;FOLD LIN P827 Vel=2 m/s CPDAT827 Tool[1]:marker Base[0] ;%{PE}
;FOLD Parameters ;%{h}
;Params IlfProvider=kukaroboter.basistech.inlineforms.movement.old; Kuka.IsGlobalPoint=False; Kuka.PointName=P827; Kuka.BlendingEnabled=False; Kuka.MoveDataName=CPDAT1; Kuka.VelocityPath=2; Kuka.CurrentCDSetIndex=0; Kuka.MovementParameterFieldEnabled=True; IlfCommand=LIN
;ENDFOLD
$BWDSTART = FALSE
LDAT_ACT = LCPDAT827
FDAT_ACT = FP827
BAS(#CP_PARAMS, 2.0)
SET_CD_PARAMS (0)
LIN XP827
;ENDFOLD

;FOLD LIN P828 Vel=2 m/s CPDAT828 Tool[1]:marker Base[0] ;%{PE}
;FOLD Parameters ;%{h}
;Params IlfProvider=kukaroboter.basistech.inlineforms.movement.old; Kuka.IsGlobalPoint=False; Kuka.PointName=P828; Kuka.BlendingEnabled=False; Kuka.MoveDataName=CPDAT1; Kuka.VelocityPath=2; Kuka.CurrentCDSetIndex=0; Kuka.MovementParameterFieldEnabled=True; IlfCommand=LIN
;ENDFOLD
$BWDSTART = FALSE
LDAT_ACT = LCPDAT828
FDAT_ACT = FP828
BAS(#CP_PARAMS, 2.0)
SET_CD_PARAMS (0)
LIN XP828
;ENDFOLD

;FOLD LIN P829 Vel=2 m/s CPDAT829 Tool[1]:marker Base[0] ;%{PE}
;FOLD Parameters ;%{h}
;Params IlfProvider=kukaroboter.basistech.inlineforms.movement.old; Kuka.IsGlobalPoint=False; Kuka.PointName=P829; Kuka.BlendingEnabled=False; Kuka.MoveDataName=CPDAT1; Kuka.VelocityPath=2; Kuka.CurrentCDSetIndex=0; Kuka.MovementParameterFieldEnabled=True; IlfCommand=LIN
;ENDFOLD
$BWDSTART = FALSE
LDAT_ACT = LCPDAT829
FDAT_ACT = FP829
BAS(#CP_PARAMS, 2.0)
SET_CD_PARAMS (0)
LIN XP829
;ENDFOLD

;FOLD LIN P830 Vel=2 m/s CPDAT830 Tool[1]:marker Base[0] ;%{PE}
;FOLD Parameters ;%{h}
;Params IlfProvider=kukaroboter.basistech.inlineforms.movement.old; Kuka.IsGlobalPoint=False; Kuka.PointName=P830; Kuka.BlendingEnabled=False; Kuka.MoveDataName=CPDAT1; Kuka.VelocityPath=2; Kuka.CurrentCDSetIndex=0; Kuka.MovementParameterFieldEnabled=True; IlfCommand=LIN
;ENDFOLD
$BWDSTART = FALSE
LDAT_ACT = LCPDAT830
FDAT_ACT = FP830
BAS(#CP_PARAMS, 2.0)
SET_CD_PARAMS (0)
LIN XP830
;ENDFOLD

;FOLD LIN P831 Vel=2 m/s CPDAT831 Tool[1]:marker Base[0] ;%{PE}
;FOLD Parameters ;%{h}
;Params IlfProvider=kukaroboter.basistech.inlineforms.movement.old; Kuka.IsGlobalPoint=False; Kuka.PointName=P831; Kuka.BlendingEnabled=False; Kuka.MoveDataName=CPDAT1; Kuka.VelocityPath=2; Kuka.CurrentCDSetIndex=0; Kuka.MovementParameterFieldEnabled=True; IlfCommand=LIN
;ENDFOLD
$BWDSTART = FALSE
LDAT_ACT = LCPDAT831
FDAT_ACT = FP831
BAS(#CP_PARAMS, 2.0)
SET_CD_PARAMS (0)
LIN XP831
;ENDFOLD

;FOLD LIN P832 Vel=2 m/s CPDAT832 Tool[1]:marker Base[0] ;%{PE}
;FOLD Parameters ;%{h}
;Params IlfProvider=kukaroboter.basistech.inlineforms.movement.old; Kuka.IsGlobalPoint=False; Kuka.PointName=P832; Kuka.BlendingEnabled=False; Kuka.MoveDataName=CPDAT1; Kuka.VelocityPath=2; Kuka.CurrentCDSetIndex=0; Kuka.MovementParameterFieldEnabled=True; IlfCommand=LIN
;ENDFOLD
$BWDSTART = FALSE
LDAT_ACT = LCPDAT832
FDAT_ACT = FP832
BAS(#CP_PARAMS, 2.0)
SET_CD_PARAMS (0)
LIN XP832
;ENDFOLD

;FOLD LIN P833 Vel=2 m/s CPDAT833 Tool[1]:marker Base[0] ;%{PE}
;FOLD Parameters ;%{h}
;Params IlfProvider=kukaroboter.basistech.inlineforms.movement.old; Kuka.IsGlobalPoint=False; Kuka.PointName=P833; Kuka.BlendingEnabled=False; Kuka.MoveDataName=CPDAT1; Kuka.VelocityPath=2; Kuka.CurrentCDSetIndex=0; Kuka.MovementParameterFieldEnabled=True; IlfCommand=LIN
;ENDFOLD
$BWDSTART = FALSE
LDAT_ACT = LCPDAT833
FDAT_ACT = FP833
BAS(#CP_PARAMS, 2.0)
SET_CD_PARAMS (0)
LIN XP833
;ENDFOLD

;FOLD LIN P834 Vel=2 m/s CPDAT834 Tool[1]:marker Base[0] ;%{PE}
;FOLD Parameters ;%{h}
;Params IlfProvider=kukaroboter.basistech.inlineforms.movement.old; Kuka.IsGlobalPoint=False; Kuka.PointName=P834; Kuka.BlendingEnabled=False; Kuka.MoveDataName=CPDAT1; Kuka.VelocityPath=2; Kuka.CurrentCDSetIndex=0; Kuka.MovementParameterFieldEnabled=True; IlfCommand=LIN
;ENDFOLD
$BWDSTART = FALSE
LDAT_ACT = LCPDAT834
FDAT_ACT = FP834
BAS(#CP_PARAMS, 2.0)
SET_CD_PARAMS (0)
LIN XP834
;ENDFOLD

;FOLD LIN P835 Vel=2 m/s CPDAT835 Tool[1]:marker Base[0] ;%{PE}
;FOLD Parameters ;%{h}
;Params IlfProvider=kukaroboter.basistech.inlineforms.movement.old; Kuka.IsGlobalPoint=False; Kuka.PointName=P835; Kuka.BlendingEnabled=False; Kuka.MoveDataName=CPDAT1; Kuka.VelocityPath=2; Kuka.CurrentCDSetIndex=0; Kuka.MovementParameterFieldEnabled=True; IlfCommand=LIN
;ENDFOLD
$BWDSTART = FALSE
LDAT_ACT = LCPDAT835
FDAT_ACT = FP835
BAS(#CP_PARAMS, 2.0)
SET_CD_PARAMS (0)
LIN XP835
;ENDFOLD

;FOLD LIN P836 Vel=2 m/s CPDAT836 Tool[1]:marker Base[0] ;%{PE}
;FOLD Parameters ;%{h}
;Params IlfProvider=kukaroboter.basistech.inlineforms.movement.old; Kuka.IsGlobalPoint=False; Kuka.PointName=P836; Kuka.BlendingEnabled=False; Kuka.MoveDataName=CPDAT1; Kuka.VelocityPath=2; Kuka.CurrentCDSetIndex=0; Kuka.MovementParameterFieldEnabled=True; IlfCommand=LIN
;ENDFOLD
$BWDSTART = FALSE
LDAT_ACT = LCPDAT836
FDAT_ACT = FP836
BAS(#CP_PARAMS, 2.0)
SET_CD_PARAMS (0)
LIN XP836
;ENDFOLD

;FOLD LIN P837 Vel=2 m/s CPDAT837 Tool[1]:marker Base[0] ;%{PE}
;FOLD Parameters ;%{h}
;Params IlfProvider=kukaroboter.basistech.inlineforms.movement.old; Kuka.IsGlobalPoint=False; Kuka.PointName=P837; Kuka.BlendingEnabled=False; Kuka.MoveDataName=CPDAT1; Kuka.VelocityPath=2; Kuka.CurrentCDSetIndex=0; Kuka.MovementParameterFieldEnabled=True; IlfCommand=LIN
;ENDFOLD
$BWDSTART = FALSE
LDAT_ACT = LCPDAT837
FDAT_ACT = FP837
BAS(#CP_PARAMS, 2.0)
SET_CD_PARAMS (0)
LIN XP837
;ENDFOLD

;FOLD LIN P838 Vel=2 m/s CPDAT838 Tool[1]:marker Base[0] ;%{PE}
;FOLD Parameters ;%{h}
;Params IlfProvider=kukaroboter.basistech.inlineforms.movement.old; Kuka.IsGlobalPoint=False; Kuka.PointName=P838; Kuka.BlendingEnabled=False; Kuka.MoveDataName=CPDAT1; Kuka.VelocityPath=2; Kuka.CurrentCDSetIndex=0; Kuka.MovementParameterFieldEnabled=True; IlfCommand=LIN
;ENDFOLD
$BWDSTART = FALSE
LDAT_ACT = LCPDAT838
FDAT_ACT = FP838
BAS(#CP_PARAMS, 2.0)
SET_CD_PARAMS (0)
LIN XP838
;ENDFOLD

;FOLD LIN P839 Vel=2 m/s CPDAT839 Tool[1]:marker Base[0] ;%{PE}
;FOLD Parameters ;%{h}
;Params IlfProvider=kukaroboter.basistech.inlineforms.movement.old; Kuka.IsGlobalPoint=False; Kuka.PointName=P839; Kuka.BlendingEnabled=False; Kuka.MoveDataName=CPDAT1; Kuka.VelocityPath=2; Kuka.CurrentCDSetIndex=0; Kuka.MovementParameterFieldEnabled=True; IlfCommand=LIN
;ENDFOLD
$BWDSTART = FALSE
LDAT_ACT = LCPDAT839
FDAT_ACT = FP839
BAS(#CP_PARAMS, 2.0)
SET_CD_PARAMS (0)
LIN XP839
;ENDFOLD

;FOLD LIN P840 Vel=2 m/s CPDAT840 Tool[1]:marker Base[0] ;%{PE}
;FOLD Parameters ;%{h}
;Params IlfProvider=kukaroboter.basistech.inlineforms.movement.old; Kuka.IsGlobalPoint=False; Kuka.PointName=P840; Kuka.BlendingEnabled=False; Kuka.MoveDataName=CPDAT1; Kuka.VelocityPath=2; Kuka.CurrentCDSetIndex=0; Kuka.MovementParameterFieldEnabled=True; IlfCommand=LIN
;ENDFOLD
$BWDSTART = FALSE
LDAT_ACT = LCPDAT840
FDAT_ACT = FP840
BAS(#CP_PARAMS, 2.0)
SET_CD_PARAMS (0)
LIN XP840
;ENDFOLD

;FOLD LIN P841 Vel=2 m/s CPDAT841 Tool[1]:marker Base[0] ;%{PE}
;FOLD Parameters ;%{h}
;Params IlfProvider=kukaroboter.basistech.inlineforms.movement.old; Kuka.IsGlobalPoint=False; Kuka.PointName=P841; Kuka.BlendingEnabled=False; Kuka.MoveDataName=CPDAT1; Kuka.VelocityPath=2; Kuka.CurrentCDSetIndex=0; Kuka.MovementParameterFieldEnabled=True; IlfCommand=LIN
;ENDFOLD
$BWDSTART = FALSE
LDAT_ACT = LCPDAT841
FDAT_ACT = FP841
BAS(#CP_PARAMS, 2.0)
SET_CD_PARAMS (0)
LIN XP841
;ENDFOLD

;FOLD LIN P842 Vel=2 m/s CPDAT842 Tool[1]:marker Base[0] ;%{PE}
;FOLD Parameters ;%{h}
;Params IlfProvider=kukaroboter.basistech.inlineforms.movement.old; Kuka.IsGlobalPoint=False; Kuka.PointName=P842; Kuka.BlendingEnabled=False; Kuka.MoveDataName=CPDAT1; Kuka.VelocityPath=2; Kuka.CurrentCDSetIndex=0; Kuka.MovementParameterFieldEnabled=True; IlfCommand=LIN
;ENDFOLD
$BWDSTART = FALSE
LDAT_ACT = LCPDAT842
FDAT_ACT = FP842
BAS(#CP_PARAMS, 2.0)
SET_CD_PARAMS (0)
LIN XP842
;ENDFOLD

;FOLD LIN P843 Vel=2 m/s CPDAT843 Tool[1]:marker Base[0] ;%{PE}
;FOLD Parameters ;%{h}
;Params IlfProvider=kukaroboter.basistech.inlineforms.movement.old; Kuka.IsGlobalPoint=False; Kuka.PointName=P843; Kuka.BlendingEnabled=False; Kuka.MoveDataName=CPDAT1; Kuka.VelocityPath=2; Kuka.CurrentCDSetIndex=0; Kuka.MovementParameterFieldEnabled=True; IlfCommand=LIN
;ENDFOLD
$BWDSTART = FALSE
LDAT_ACT = LCPDAT843
FDAT_ACT = FP843
BAS(#CP_PARAMS, 2.0)
SET_CD_PARAMS (0)
LIN XP843
;ENDFOLD

;FOLD LIN P844 Vel=2 m/s CPDAT844 Tool[1]:marker Base[0] ;%{PE}
;FOLD Parameters ;%{h}
;Params IlfProvider=kukaroboter.basistech.inlineforms.movement.old; Kuka.IsGlobalPoint=False; Kuka.PointName=P844; Kuka.BlendingEnabled=False; Kuka.MoveDataName=CPDAT1; Kuka.VelocityPath=2; Kuka.CurrentCDSetIndex=0; Kuka.MovementParameterFieldEnabled=True; IlfCommand=LIN
;ENDFOLD
$BWDSTART = FALSE
LDAT_ACT = LCPDAT844
FDAT_ACT = FP844
BAS(#CP_PARAMS, 2.0)
SET_CD_PARAMS (0)
LIN XP844
;ENDFOLD

;FOLD LIN P845 Vel=2 m/s CPDAT845 Tool[1]:marker Base[0] ;%{PE}
;FOLD Parameters ;%{h}
;Params IlfProvider=kukaroboter.basistech.inlineforms.movement.old; Kuka.IsGlobalPoint=False; Kuka.PointName=P845; Kuka.BlendingEnabled=False; Kuka.MoveDataName=CPDAT1; Kuka.VelocityPath=2; Kuka.CurrentCDSetIndex=0; Kuka.MovementParameterFieldEnabled=True; IlfCommand=LIN
;ENDFOLD
$BWDSTART = FALSE
LDAT_ACT = LCPDAT845
FDAT_ACT = FP845
BAS(#CP_PARAMS, 2.0)
SET_CD_PARAMS (0)
LIN XP845
;ENDFOLD

;FOLD LIN P846 Vel=2 m/s CPDAT846 Tool[1]:marker Base[0] ;%{PE}
;FOLD Parameters ;%{h}
;Params IlfProvider=kukaroboter.basistech.inlineforms.movement.old; Kuka.IsGlobalPoint=False; Kuka.PointName=P846; Kuka.BlendingEnabled=False; Kuka.MoveDataName=CPDAT1; Kuka.VelocityPath=2; Kuka.CurrentCDSetIndex=0; Kuka.MovementParameterFieldEnabled=True; IlfCommand=LIN
;ENDFOLD
$BWDSTART = FALSE
LDAT_ACT = LCPDAT846
FDAT_ACT = FP846
BAS(#CP_PARAMS, 2.0)
SET_CD_PARAMS (0)
LIN XP846
;ENDFOLD

;FOLD LIN P847 Vel=2 m/s CPDAT847 Tool[1]:marker Base[0] ;%{PE}
;FOLD Parameters ;%{h}
;Params IlfProvider=kukaroboter.basistech.inlineforms.movement.old; Kuka.IsGlobalPoint=False; Kuka.PointName=P847; Kuka.BlendingEnabled=False; Kuka.MoveDataName=CPDAT1; Kuka.VelocityPath=2; Kuka.CurrentCDSetIndex=0; Kuka.MovementParameterFieldEnabled=True; IlfCommand=LIN
;ENDFOLD
$BWDSTART = FALSE
LDAT_ACT = LCPDAT847
FDAT_ACT = FP847
BAS(#CP_PARAMS, 2.0)
SET_CD_PARAMS (0)
LIN XP847
;ENDFOLD

;FOLD LIN P848 Vel=2 m/s CPDAT848 Tool[1]:marker Base[0] ;%{PE}
;FOLD Parameters ;%{h}
;Params IlfProvider=kukaroboter.basistech.inlineforms.movement.old; Kuka.IsGlobalPoint=False; Kuka.PointName=P848; Kuka.BlendingEnabled=False; Kuka.MoveDataName=CPDAT1; Kuka.VelocityPath=2; Kuka.CurrentCDSetIndex=0; Kuka.MovementParameterFieldEnabled=True; IlfCommand=LIN
;ENDFOLD
$BWDSTART = FALSE
LDAT_ACT = LCPDAT848
FDAT_ACT = FP848
BAS(#CP_PARAMS, 2.0)
SET_CD_PARAMS (0)
LIN XP848
;ENDFOLD

;FOLD LIN P849 Vel=2 m/s CPDAT849 Tool[1]:marker Base[0] ;%{PE}
;FOLD Parameters ;%{h}
;Params IlfProvider=kukaroboter.basistech.inlineforms.movement.old; Kuka.IsGlobalPoint=False; Kuka.PointName=P849; Kuka.BlendingEnabled=False; Kuka.MoveDataName=CPDAT1; Kuka.VelocityPath=2; Kuka.CurrentCDSetIndex=0; Kuka.MovementParameterFieldEnabled=True; IlfCommand=LIN
;ENDFOLD
$BWDSTART = FALSE
LDAT_ACT = LCPDAT849
FDAT_ACT = FP849
BAS(#CP_PARAMS, 2.0)
SET_CD_PARAMS (0)
LIN XP849
;ENDFOLD

;FOLD LIN P850 Vel=2 m/s CPDAT850 Tool[1]:marker Base[0] ;%{PE}
;FOLD Parameters ;%{h}
;Params IlfProvider=kukaroboter.basistech.inlineforms.movement.old; Kuka.IsGlobalPoint=False; Kuka.PointName=P850; Kuka.BlendingEnabled=False; Kuka.MoveDataName=CPDAT1; Kuka.VelocityPath=2; Kuka.CurrentCDSetIndex=0; Kuka.MovementParameterFieldEnabled=True; IlfCommand=LIN
;ENDFOLD
$BWDSTART = FALSE
LDAT_ACT = LCPDAT850
FDAT_ACT = FP850
BAS(#CP_PARAMS, 2.0)
SET_CD_PARAMS (0)
LIN XP850
;ENDFOLD

;FOLD LIN P851 Vel=2 m/s CPDAT851 Tool[1]:marker Base[0] ;%{PE}
;FOLD Parameters ;%{h}
;Params IlfProvider=kukaroboter.basistech.inlineforms.movement.old; Kuka.IsGlobalPoint=False; Kuka.PointName=P851; Kuka.BlendingEnabled=False; Kuka.MoveDataName=CPDAT1; Kuka.VelocityPath=2; Kuka.CurrentCDSetIndex=0; Kuka.MovementParameterFieldEnabled=True; IlfCommand=LIN
;ENDFOLD
$BWDSTART = FALSE
LDAT_ACT = LCPDAT851
FDAT_ACT = FP851
BAS(#CP_PARAMS, 2.0)
SET_CD_PARAMS (0)
LIN XP851
;ENDFOLD

;FOLD LIN P852 Vel=2 m/s CPDAT852 Tool[1]:marker Base[0] ;%{PE}
;FOLD Parameters ;%{h}
;Params IlfProvider=kukaroboter.basistech.inlineforms.movement.old; Kuka.IsGlobalPoint=False; Kuka.PointName=P852; Kuka.BlendingEnabled=False; Kuka.MoveDataName=CPDAT1; Kuka.VelocityPath=2; Kuka.CurrentCDSetIndex=0; Kuka.MovementParameterFieldEnabled=True; IlfCommand=LIN
;ENDFOLD
$BWDSTART = FALSE
LDAT_ACT = LCPDAT852
FDAT_ACT = FP852
BAS(#CP_PARAMS, 2.0)
SET_CD_PARAMS (0)
LIN XP852
;ENDFOLD

;FOLD LIN P853 Vel=2 m/s CPDAT853 Tool[1]:marker Base[0] ;%{PE}
;FOLD Parameters ;%{h}
;Params IlfProvider=kukaroboter.basistech.inlineforms.movement.old; Kuka.IsGlobalPoint=False; Kuka.PointName=P853; Kuka.BlendingEnabled=False; Kuka.MoveDataName=CPDAT1; Kuka.VelocityPath=2; Kuka.CurrentCDSetIndex=0; Kuka.MovementParameterFieldEnabled=True; IlfCommand=LIN
;ENDFOLD
$BWDSTART = FALSE
LDAT_ACT = LCPDAT853
FDAT_ACT = FP853
BAS(#CP_PARAMS, 2.0)
SET_CD_PARAMS (0)
LIN XP853
;ENDFOLD

;FOLD LIN P854 Vel=2 m/s CPDAT854 Tool[1]:marker Base[0] ;%{PE}
;FOLD Parameters ;%{h}
;Params IlfProvider=kukaroboter.basistech.inlineforms.movement.old; Kuka.IsGlobalPoint=False; Kuka.PointName=P854; Kuka.BlendingEnabled=False; Kuka.MoveDataName=CPDAT1; Kuka.VelocityPath=2; Kuka.CurrentCDSetIndex=0; Kuka.MovementParameterFieldEnabled=True; IlfCommand=LIN
;ENDFOLD
$BWDSTART = FALSE
LDAT_ACT = LCPDAT854
FDAT_ACT = FP854
BAS(#CP_PARAMS, 2.0)
SET_CD_PARAMS (0)
LIN XP854
;ENDFOLD

;FOLD LIN P855 Vel=2 m/s CPDAT855 Tool[1]:marker Base[0] ;%{PE}
;FOLD Parameters ;%{h}
;Params IlfProvider=kukaroboter.basistech.inlineforms.movement.old; Kuka.IsGlobalPoint=False; Kuka.PointName=P855; Kuka.BlendingEnabled=False; Kuka.MoveDataName=CPDAT1; Kuka.VelocityPath=2; Kuka.CurrentCDSetIndex=0; Kuka.MovementParameterFieldEnabled=True; IlfCommand=LIN
;ENDFOLD
$BWDSTART = FALSE
LDAT_ACT = LCPDAT855
FDAT_ACT = FP855
BAS(#CP_PARAMS, 2.0)
SET_CD_PARAMS (0)
LIN XP855
;ENDFOLD

;FOLD LIN P856 Vel=2 m/s CPDAT856 Tool[1]:marker Base[0] ;%{PE}
;FOLD Parameters ;%{h}
;Params IlfProvider=kukaroboter.basistech.inlineforms.movement.old; Kuka.IsGlobalPoint=False; Kuka.PointName=P856; Kuka.BlendingEnabled=False; Kuka.MoveDataName=CPDAT1; Kuka.VelocityPath=2; Kuka.CurrentCDSetIndex=0; Kuka.MovementParameterFieldEnabled=True; IlfCommand=LIN
;ENDFOLD
$BWDSTART = FALSE
LDAT_ACT = LCPDAT856
FDAT_ACT = FP856
BAS(#CP_PARAMS, 2.0)
SET_CD_PARAMS (0)
LIN XP856
;ENDFOLD

;FOLD LIN P857 Vel=2 m/s CPDAT857 Tool[1]:marker Base[0] ;%{PE}
;FOLD Parameters ;%{h}
;Params IlfProvider=kukaroboter.basistech.inlineforms.movement.old; Kuka.IsGlobalPoint=False; Kuka.PointName=P857; Kuka.BlendingEnabled=False; Kuka.MoveDataName=CPDAT1; Kuka.VelocityPath=2; Kuka.CurrentCDSetIndex=0; Kuka.MovementParameterFieldEnabled=True; IlfCommand=LIN
;ENDFOLD
$BWDSTART = FALSE
LDAT_ACT = LCPDAT857
FDAT_ACT = FP857
BAS(#CP_PARAMS, 2.0)
SET_CD_PARAMS (0)
LIN XP857
;ENDFOLD

;FOLD LIN P858 Vel=2 m/s CPDAT858 Tool[1]:marker Base[0] ;%{PE}
;FOLD Parameters ;%{h}
;Params IlfProvider=kukaroboter.basistech.inlineforms.movement.old; Kuka.IsGlobalPoint=False; Kuka.PointName=P858; Kuka.BlendingEnabled=False; Kuka.MoveDataName=CPDAT1; Kuka.VelocityPath=2; Kuka.CurrentCDSetIndex=0; Kuka.MovementParameterFieldEnabled=True; IlfCommand=LIN
;ENDFOLD
$BWDSTART = FALSE
LDAT_ACT = LCPDAT858
FDAT_ACT = FP858
BAS(#CP_PARAMS, 2.0)
SET_CD_PARAMS (0)
LIN XP858
;ENDFOLD

;FOLD LIN P859 Vel=2 m/s CPDAT859 Tool[1]:marker Base[0] ;%{PE}
;FOLD Parameters ;%{h}
;Params IlfProvider=kukaroboter.basistech.inlineforms.movement.old; Kuka.IsGlobalPoint=False; Kuka.PointName=P859; Kuka.BlendingEnabled=False; Kuka.MoveDataName=CPDAT1; Kuka.VelocityPath=2; Kuka.CurrentCDSetIndex=0; Kuka.MovementParameterFieldEnabled=True; IlfCommand=LIN
;ENDFOLD
$BWDSTART = FALSE
LDAT_ACT = LCPDAT859
FDAT_ACT = FP859
BAS(#CP_PARAMS, 2.0)
SET_CD_PARAMS (0)
LIN XP859
;ENDFOLD

;FOLD LIN P860 Vel=2 m/s CPDAT860 Tool[1]:marker Base[0] ;%{PE}
;FOLD Parameters ;%{h}
;Params IlfProvider=kukaroboter.basistech.inlineforms.movement.old; Kuka.IsGlobalPoint=False; Kuka.PointName=P860; Kuka.BlendingEnabled=False; Kuka.MoveDataName=CPDAT1; Kuka.VelocityPath=2; Kuka.CurrentCDSetIndex=0; Kuka.MovementParameterFieldEnabled=True; IlfCommand=LIN
;ENDFOLD
$BWDSTART = FALSE
LDAT_ACT = LCPDAT860
FDAT_ACT = FP860
BAS(#CP_PARAMS, 2.0)
SET_CD_PARAMS (0)
LIN XP860
;ENDFOLD

;FOLD LIN P861 Vel=2 m/s CPDAT861 Tool[1]:marker Base[0] ;%{PE}
;FOLD Parameters ;%{h}
;Params IlfProvider=kukaroboter.basistech.inlineforms.movement.old; Kuka.IsGlobalPoint=False; Kuka.PointName=P861; Kuka.BlendingEnabled=False; Kuka.MoveDataName=CPDAT1; Kuka.VelocityPath=2; Kuka.CurrentCDSetIndex=0; Kuka.MovementParameterFieldEnabled=True; IlfCommand=LIN
;ENDFOLD
$BWDSTART = FALSE
LDAT_ACT = LCPDAT861
FDAT_ACT = FP861
BAS(#CP_PARAMS, 2.0)
SET_CD_PARAMS (0)
LIN XP861
;ENDFOLD

;FOLD LIN P862 Vel=2 m/s CPDAT862 Tool[1]:marker Base[0] ;%{PE}
;FOLD Parameters ;%{h}
;Params IlfProvider=kukaroboter.basistech.inlineforms.movement.old; Kuka.IsGlobalPoint=False; Kuka.PointName=P862; Kuka.BlendingEnabled=False; Kuka.MoveDataName=CPDAT1; Kuka.VelocityPath=2; Kuka.CurrentCDSetIndex=0; Kuka.MovementParameterFieldEnabled=True; IlfCommand=LIN
;ENDFOLD
$BWDSTART = FALSE
LDAT_ACT = LCPDAT862
FDAT_ACT = FP862
BAS(#CP_PARAMS, 2.0)
SET_CD_PARAMS (0)
LIN XP862
;ENDFOLD

;FOLD LIN P863 Vel=2 m/s CPDAT863 Tool[1]:marker Base[0] ;%{PE}
;FOLD Parameters ;%{h}
;Params IlfProvider=kukaroboter.basistech.inlineforms.movement.old; Kuka.IsGlobalPoint=False; Kuka.PointName=P863; Kuka.BlendingEnabled=False; Kuka.MoveDataName=CPDAT1; Kuka.VelocityPath=2; Kuka.CurrentCDSetIndex=0; Kuka.MovementParameterFieldEnabled=True; IlfCommand=LIN
;ENDFOLD
$BWDSTART = FALSE
LDAT_ACT = LCPDAT863
FDAT_ACT = FP863
BAS(#CP_PARAMS, 2.0)
SET_CD_PARAMS (0)
LIN XP863
;ENDFOLD

;FOLD LIN P864 Vel=2 m/s CPDAT864 Tool[1]:marker Base[0] ;%{PE}
;FOLD Parameters ;%{h}
;Params IlfProvider=kukaroboter.basistech.inlineforms.movement.old; Kuka.IsGlobalPoint=False; Kuka.PointName=P864; Kuka.BlendingEnabled=False; Kuka.MoveDataName=CPDAT1; Kuka.VelocityPath=2; Kuka.CurrentCDSetIndex=0; Kuka.MovementParameterFieldEnabled=True; IlfCommand=LIN
;ENDFOLD
$BWDSTART = FALSE
LDAT_ACT = LCPDAT864
FDAT_ACT = FP864
BAS(#CP_PARAMS, 2.0)
SET_CD_PARAMS (0)
LIN XP864
;ENDFOLD

;FOLD LIN P865 Vel=2 m/s CPDAT865 Tool[1]:marker Base[0] ;%{PE}
;FOLD Parameters ;%{h}
;Params IlfProvider=kukaroboter.basistech.inlineforms.movement.old; Kuka.IsGlobalPoint=False; Kuka.PointName=P865; Kuka.BlendingEnabled=False; Kuka.MoveDataName=CPDAT1; Kuka.VelocityPath=2; Kuka.CurrentCDSetIndex=0; Kuka.MovementParameterFieldEnabled=True; IlfCommand=LIN
;ENDFOLD
$BWDSTART = FALSE
LDAT_ACT = LCPDAT865
FDAT_ACT = FP865
BAS(#CP_PARAMS, 2.0)
SET_CD_PARAMS (0)
LIN XP865
;ENDFOLD

;FOLD LIN P866 Vel=2 m/s CPDAT866 Tool[1]:marker Base[0] ;%{PE}
;FOLD Parameters ;%{h}
;Params IlfProvider=kukaroboter.basistech.inlineforms.movement.old; Kuka.IsGlobalPoint=False; Kuka.PointName=P866; Kuka.BlendingEnabled=False; Kuka.MoveDataName=CPDAT1; Kuka.VelocityPath=2; Kuka.CurrentCDSetIndex=0; Kuka.MovementParameterFieldEnabled=True; IlfCommand=LIN
;ENDFOLD
$BWDSTART = FALSE
LDAT_ACT = LCPDAT866
FDAT_ACT = FP866
BAS(#CP_PARAMS, 2.0)
SET_CD_PARAMS (0)
LIN XP866
;ENDFOLD

;FOLD LIN P867 Vel=2 m/s CPDAT867 Tool[1]:marker Base[0] ;%{PE}
;FOLD Parameters ;%{h}
;Params IlfProvider=kukaroboter.basistech.inlineforms.movement.old; Kuka.IsGlobalPoint=False; Kuka.PointName=P867; Kuka.BlendingEnabled=False; Kuka.MoveDataName=CPDAT1; Kuka.VelocityPath=2; Kuka.CurrentCDSetIndex=0; Kuka.MovementParameterFieldEnabled=True; IlfCommand=LIN
;ENDFOLD
$BWDSTART = FALSE
LDAT_ACT = LCPDAT867
FDAT_ACT = FP867
BAS(#CP_PARAMS, 2.0)
SET_CD_PARAMS (0)
LIN XP867
;ENDFOLD

;FOLD LIN P868 Vel=2 m/s CPDAT868 Tool[1]:marker Base[0] ;%{PE}
;FOLD Parameters ;%{h}
;Params IlfProvider=kukaroboter.basistech.inlineforms.movement.old; Kuka.IsGlobalPoint=False; Kuka.PointName=P868; Kuka.BlendingEnabled=False; Kuka.MoveDataName=CPDAT1; Kuka.VelocityPath=2; Kuka.CurrentCDSetIndex=0; Kuka.MovementParameterFieldEnabled=True; IlfCommand=LIN
;ENDFOLD
$BWDSTART = FALSE
LDAT_ACT = LCPDAT868
FDAT_ACT = FP868
BAS(#CP_PARAMS, 2.0)
SET_CD_PARAMS (0)
LIN XP868
;ENDFOLD

;FOLD LIN P869 Vel=2 m/s CPDAT869 Tool[1]:marker Base[0] ;%{PE}
;FOLD Parameters ;%{h}
;Params IlfProvider=kukaroboter.basistech.inlineforms.movement.old; Kuka.IsGlobalPoint=False; Kuka.PointName=P869; Kuka.BlendingEnabled=False; Kuka.MoveDataName=CPDAT1; Kuka.VelocityPath=2; Kuka.CurrentCDSetIndex=0; Kuka.MovementParameterFieldEnabled=True; IlfCommand=LIN
;ENDFOLD
$BWDSTART = FALSE
LDAT_ACT = LCPDAT869
FDAT_ACT = FP869
BAS(#CP_PARAMS, 2.0)
SET_CD_PARAMS (0)
LIN XP869
;ENDFOLD

;FOLD LIN P870 Vel=2 m/s CPDAT870 Tool[1]:marker Base[0] ;%{PE}
;FOLD Parameters ;%{h}
;Params IlfProvider=kukaroboter.basistech.inlineforms.movement.old; Kuka.IsGlobalPoint=False; Kuka.PointName=P870; Kuka.BlendingEnabled=False; Kuka.MoveDataName=CPDAT1; Kuka.VelocityPath=2; Kuka.CurrentCDSetIndex=0; Kuka.MovementParameterFieldEnabled=True; IlfCommand=LIN
;ENDFOLD
$BWDSTART = FALSE
LDAT_ACT = LCPDAT870
FDAT_ACT = FP870
BAS(#CP_PARAMS, 2.0)
SET_CD_PARAMS (0)
LIN XP870
;ENDFOLD

;FOLD LIN P871 Vel=2 m/s CPDAT871 Tool[1]:marker Base[0] ;%{PE}
;FOLD Parameters ;%{h}
;Params IlfProvider=kukaroboter.basistech.inlineforms.movement.old; Kuka.IsGlobalPoint=False; Kuka.PointName=P871; Kuka.BlendingEnabled=False; Kuka.MoveDataName=CPDAT1; Kuka.VelocityPath=2; Kuka.CurrentCDSetIndex=0; Kuka.MovementParameterFieldEnabled=True; IlfCommand=LIN
;ENDFOLD
$BWDSTART = FALSE
LDAT_ACT = LCPDAT871
FDAT_ACT = FP871
BAS(#CP_PARAMS, 2.0)
SET_CD_PARAMS (0)
LIN XP871
;ENDFOLD

;FOLD LIN P872 Vel=2 m/s CPDAT872 Tool[1]:marker Base[0] ;%{PE}
;FOLD Parameters ;%{h}
;Params IlfProvider=kukaroboter.basistech.inlineforms.movement.old; Kuka.IsGlobalPoint=False; Kuka.PointName=P872; Kuka.BlendingEnabled=False; Kuka.MoveDataName=CPDAT1; Kuka.VelocityPath=2; Kuka.CurrentCDSetIndex=0; Kuka.MovementParameterFieldEnabled=True; IlfCommand=LIN
;ENDFOLD
$BWDSTART = FALSE
LDAT_ACT = LCPDAT872
FDAT_ACT = FP872
BAS(#CP_PARAMS, 2.0)
SET_CD_PARAMS (0)
LIN XP872
;ENDFOLD

;FOLD LIN P873 Vel=2 m/s CPDAT873 Tool[1]:marker Base[0] ;%{PE}
;FOLD Parameters ;%{h}
;Params IlfProvider=kukaroboter.basistech.inlineforms.movement.old; Kuka.IsGlobalPoint=False; Kuka.PointName=P873; Kuka.BlendingEnabled=False; Kuka.MoveDataName=CPDAT1; Kuka.VelocityPath=2; Kuka.CurrentCDSetIndex=0; Kuka.MovementParameterFieldEnabled=True; IlfCommand=LIN
;ENDFOLD
$BWDSTART = FALSE
LDAT_ACT = LCPDAT873
FDAT_ACT = FP873
BAS(#CP_PARAMS, 2.0)
SET_CD_PARAMS (0)
LIN XP873
;ENDFOLD

;FOLD LIN P874 Vel=2 m/s CPDAT874 Tool[1]:marker Base[0] ;%{PE}
;FOLD Parameters ;%{h}
;Params IlfProvider=kukaroboter.basistech.inlineforms.movement.old; Kuka.IsGlobalPoint=False; Kuka.PointName=P874; Kuka.BlendingEnabled=False; Kuka.MoveDataName=CPDAT1; Kuka.VelocityPath=2; Kuka.CurrentCDSetIndex=0; Kuka.MovementParameterFieldEnabled=True; IlfCommand=LIN
;ENDFOLD
$BWDSTART = FALSE
LDAT_ACT = LCPDAT874
FDAT_ACT = FP874
BAS(#CP_PARAMS, 2.0)
SET_CD_PARAMS (0)
LIN XP874
;ENDFOLD

;FOLD LIN P875 Vel=2 m/s CPDAT875 Tool[1]:marker Base[0] ;%{PE}
;FOLD Parameters ;%{h}
;Params IlfProvider=kukaroboter.basistech.inlineforms.movement.old; Kuka.IsGlobalPoint=False; Kuka.PointName=P875; Kuka.BlendingEnabled=False; Kuka.MoveDataName=CPDAT1; Kuka.VelocityPath=2; Kuka.CurrentCDSetIndex=0; Kuka.MovementParameterFieldEnabled=True; IlfCommand=LIN
;ENDFOLD
$BWDSTART = FALSE
LDAT_ACT = LCPDAT875
FDAT_ACT = FP875
BAS(#CP_PARAMS, 2.0)
SET_CD_PARAMS (0)
LIN XP875
;ENDFOLD

;FOLD LIN P876 Vel=2 m/s CPDAT876 Tool[1]:marker Base[0] ;%{PE}
;FOLD Parameters ;%{h}
;Params IlfProvider=kukaroboter.basistech.inlineforms.movement.old; Kuka.IsGlobalPoint=False; Kuka.PointName=P876; Kuka.BlendingEnabled=False; Kuka.MoveDataName=CPDAT1; Kuka.VelocityPath=2; Kuka.CurrentCDSetIndex=0; Kuka.MovementParameterFieldEnabled=True; IlfCommand=LIN
;ENDFOLD
$BWDSTART = FALSE
LDAT_ACT = LCPDAT876
FDAT_ACT = FP876
BAS(#CP_PARAMS, 2.0)
SET_CD_PARAMS (0)
LIN XP876
;ENDFOLD

;FOLD LIN P877 Vel=2 m/s CPDAT877 Tool[1]:marker Base[0] ;%{PE}
;FOLD Parameters ;%{h}
;Params IlfProvider=kukaroboter.basistech.inlineforms.movement.old; Kuka.IsGlobalPoint=False; Kuka.PointName=P877; Kuka.BlendingEnabled=False; Kuka.MoveDataName=CPDAT1; Kuka.VelocityPath=2; Kuka.CurrentCDSetIndex=0; Kuka.MovementParameterFieldEnabled=True; IlfCommand=LIN
;ENDFOLD
$BWDSTART = FALSE
LDAT_ACT = LCPDAT877
FDAT_ACT = FP877
BAS(#CP_PARAMS, 2.0)
SET_CD_PARAMS (0)
LIN XP877
;ENDFOLD

;FOLD LIN P878 Vel=2 m/s CPDAT878 Tool[1]:marker Base[0] ;%{PE}
;FOLD Parameters ;%{h}
;Params IlfProvider=kukaroboter.basistech.inlineforms.movement.old; Kuka.IsGlobalPoint=False; Kuka.PointName=P878; Kuka.BlendingEnabled=False; Kuka.MoveDataName=CPDAT1; Kuka.VelocityPath=2; Kuka.CurrentCDSetIndex=0; Kuka.MovementParameterFieldEnabled=True; IlfCommand=LIN
;ENDFOLD
$BWDSTART = FALSE
LDAT_ACT = LCPDAT878
FDAT_ACT = FP878
BAS(#CP_PARAMS, 2.0)
SET_CD_PARAMS (0)
LIN XP878
;ENDFOLD

;FOLD LIN P879 Vel=2 m/s CPDAT879 Tool[1]:marker Base[0] ;%{PE}
;FOLD Parameters ;%{h}
;Params IlfProvider=kukaroboter.basistech.inlineforms.movement.old; Kuka.IsGlobalPoint=False; Kuka.PointName=P879; Kuka.BlendingEnabled=False; Kuka.MoveDataName=CPDAT1; Kuka.VelocityPath=2; Kuka.CurrentCDSetIndex=0; Kuka.MovementParameterFieldEnabled=True; IlfCommand=LIN
;ENDFOLD
$BWDSTART = FALSE
LDAT_ACT = LCPDAT879
FDAT_ACT = FP879
BAS(#CP_PARAMS, 2.0)
SET_CD_PARAMS (0)
LIN XP879
;ENDFOLD

;FOLD LIN P880 Vel=2 m/s CPDAT880 Tool[1]:marker Base[0] ;%{PE}
;FOLD Parameters ;%{h}
;Params IlfProvider=kukaroboter.basistech.inlineforms.movement.old; Kuka.IsGlobalPoint=False; Kuka.PointName=P880; Kuka.BlendingEnabled=False; Kuka.MoveDataName=CPDAT1; Kuka.VelocityPath=2; Kuka.CurrentCDSetIndex=0; Kuka.MovementParameterFieldEnabled=True; IlfCommand=LIN
;ENDFOLD
$BWDSTART = FALSE
LDAT_ACT = LCPDAT880
FDAT_ACT = FP880
BAS(#CP_PARAMS, 2.0)
SET_CD_PARAMS (0)
LIN XP880
;ENDFOLD

;FOLD LIN P881 Vel=2 m/s CPDAT881 Tool[1]:marker Base[0] ;%{PE}
;FOLD Parameters ;%{h}
;Params IlfProvider=kukaroboter.basistech.inlineforms.movement.old; Kuka.IsGlobalPoint=False; Kuka.PointName=P881; Kuka.BlendingEnabled=False; Kuka.MoveDataName=CPDAT1; Kuka.VelocityPath=2; Kuka.CurrentCDSetIndex=0; Kuka.MovementParameterFieldEnabled=True; IlfCommand=LIN
;ENDFOLD
$BWDSTART = FALSE
LDAT_ACT = LCPDAT881
FDAT_ACT = FP881
BAS(#CP_PARAMS, 2.0)
SET_CD_PARAMS (0)
LIN XP881
;ENDFOLD

;FOLD LIN P882 Vel=2 m/s CPDAT882 Tool[1]:marker Base[0] ;%{PE}
;FOLD Parameters ;%{h}
;Params IlfProvider=kukaroboter.basistech.inlineforms.movement.old; Kuka.IsGlobalPoint=False; Kuka.PointName=P882; Kuka.BlendingEnabled=False; Kuka.MoveDataName=CPDAT1; Kuka.VelocityPath=2; Kuka.CurrentCDSetIndex=0; Kuka.MovementParameterFieldEnabled=True; IlfCommand=LIN
;ENDFOLD
$BWDSTART = FALSE
LDAT_ACT = LCPDAT882
FDAT_ACT = FP882
BAS(#CP_PARAMS, 2.0)
SET_CD_PARAMS (0)
LIN XP882
;ENDFOLD

;FOLD LIN P883 Vel=2 m/s CPDAT883 Tool[1]:marker Base[0] ;%{PE}
;FOLD Parameters ;%{h}
;Params IlfProvider=kukaroboter.basistech.inlineforms.movement.old; Kuka.IsGlobalPoint=False; Kuka.PointName=P883; Kuka.BlendingEnabled=False; Kuka.MoveDataName=CPDAT1; Kuka.VelocityPath=2; Kuka.CurrentCDSetIndex=0; Kuka.MovementParameterFieldEnabled=True; IlfCommand=LIN
;ENDFOLD
$BWDSTART = FALSE
LDAT_ACT = LCPDAT883
FDAT_ACT = FP883
BAS(#CP_PARAMS, 2.0)
SET_CD_PARAMS (0)
LIN XP883
;ENDFOLD

;FOLD LIN P884 Vel=2 m/s CPDAT884 Tool[1]:marker Base[0] ;%{PE}
;FOLD Parameters ;%{h}
;Params IlfProvider=kukaroboter.basistech.inlineforms.movement.old; Kuka.IsGlobalPoint=False; Kuka.PointName=P884; Kuka.BlendingEnabled=False; Kuka.MoveDataName=CPDAT1; Kuka.VelocityPath=2; Kuka.CurrentCDSetIndex=0; Kuka.MovementParameterFieldEnabled=True; IlfCommand=LIN
;ENDFOLD
$BWDSTART = FALSE
LDAT_ACT = LCPDAT884
FDAT_ACT = FP884
BAS(#CP_PARAMS, 2.0)
SET_CD_PARAMS (0)
LIN XP884
;ENDFOLD

;FOLD LIN P885 Vel=2 m/s CPDAT885 Tool[1]:marker Base[0] ;%{PE}
;FOLD Parameters ;%{h}
;Params IlfProvider=kukaroboter.basistech.inlineforms.movement.old; Kuka.IsGlobalPoint=False; Kuka.PointName=P885; Kuka.BlendingEnabled=False; Kuka.MoveDataName=CPDAT1; Kuka.VelocityPath=2; Kuka.CurrentCDSetIndex=0; Kuka.MovementParameterFieldEnabled=True; IlfCommand=LIN
;ENDFOLD
$BWDSTART = FALSE
LDAT_ACT = LCPDAT885
FDAT_ACT = FP885
BAS(#CP_PARAMS, 2.0)
SET_CD_PARAMS (0)
LIN XP885
;ENDFOLD

;FOLD LIN P886 Vel=2 m/s CPDAT886 Tool[1]:marker Base[0] ;%{PE}
;FOLD Parameters ;%{h}
;Params IlfProvider=kukaroboter.basistech.inlineforms.movement.old; Kuka.IsGlobalPoint=False; Kuka.PointName=P886; Kuka.BlendingEnabled=False; Kuka.MoveDataName=CPDAT1; Kuka.VelocityPath=2; Kuka.CurrentCDSetIndex=0; Kuka.MovementParameterFieldEnabled=True; IlfCommand=LIN
;ENDFOLD
$BWDSTART = FALSE
LDAT_ACT = LCPDAT886
FDAT_ACT = FP886
BAS(#CP_PARAMS, 2.0)
SET_CD_PARAMS (0)
LIN XP886
;ENDFOLD

;FOLD LIN P887 Vel=2 m/s CPDAT887 Tool[1]:marker Base[0] ;%{PE}
;FOLD Parameters ;%{h}
;Params IlfProvider=kukaroboter.basistech.inlineforms.movement.old; Kuka.IsGlobalPoint=False; Kuka.PointName=P887; Kuka.BlendingEnabled=False; Kuka.MoveDataName=CPDAT1; Kuka.VelocityPath=2; Kuka.CurrentCDSetIndex=0; Kuka.MovementParameterFieldEnabled=True; IlfCommand=LIN
;ENDFOLD
$BWDSTART = FALSE
LDAT_ACT = LCPDAT887
FDAT_ACT = FP887
BAS(#CP_PARAMS, 2.0)
SET_CD_PARAMS (0)
LIN XP887
;ENDFOLD

;FOLD LIN P888 Vel=2 m/s CPDAT888 Tool[1]:marker Base[0] ;%{PE}
;FOLD Parameters ;%{h}
;Params IlfProvider=kukaroboter.basistech.inlineforms.movement.old; Kuka.IsGlobalPoint=False; Kuka.PointName=P888; Kuka.BlendingEnabled=False; Kuka.MoveDataName=CPDAT1; Kuka.VelocityPath=2; Kuka.CurrentCDSetIndex=0; Kuka.MovementParameterFieldEnabled=True; IlfCommand=LIN
;ENDFOLD
$BWDSTART = FALSE
LDAT_ACT = LCPDAT888
FDAT_ACT = FP888
BAS(#CP_PARAMS, 2.0)
SET_CD_PARAMS (0)
LIN XP888
;ENDFOLD

;FOLD LIN P889 Vel=2 m/s CPDAT889 Tool[1]:marker Base[0] ;%{PE}
;FOLD Parameters ;%{h}
;Params IlfProvider=kukaroboter.basistech.inlineforms.movement.old; Kuka.IsGlobalPoint=False; Kuka.PointName=P889; Kuka.BlendingEnabled=False; Kuka.MoveDataName=CPDAT1; Kuka.VelocityPath=2; Kuka.CurrentCDSetIndex=0; Kuka.MovementParameterFieldEnabled=True; IlfCommand=LIN
;ENDFOLD
$BWDSTART = FALSE
LDAT_ACT = LCPDAT889
FDAT_ACT = FP889
BAS(#CP_PARAMS, 2.0)
SET_CD_PARAMS (0)
LIN XP889
;ENDFOLD

;FOLD LIN P890 Vel=2 m/s CPDAT890 Tool[1]:marker Base[0] ;%{PE}
;FOLD Parameters ;%{h}
;Params IlfProvider=kukaroboter.basistech.inlineforms.movement.old; Kuka.IsGlobalPoint=False; Kuka.PointName=P890; Kuka.BlendingEnabled=False; Kuka.MoveDataName=CPDAT1; Kuka.VelocityPath=2; Kuka.CurrentCDSetIndex=0; Kuka.MovementParameterFieldEnabled=True; IlfCommand=LIN
;ENDFOLD
$BWDSTART = FALSE
LDAT_ACT = LCPDAT890
FDAT_ACT = FP890
BAS(#CP_PARAMS, 2.0)
SET_CD_PARAMS (0)
LIN XP890
;ENDFOLD

;FOLD LIN P891 Vel=2 m/s CPDAT891 Tool[1]:marker Base[0] ;%{PE}
;FOLD Parameters ;%{h}
;Params IlfProvider=kukaroboter.basistech.inlineforms.movement.old; Kuka.IsGlobalPoint=False; Kuka.PointName=P891; Kuka.BlendingEnabled=False; Kuka.MoveDataName=CPDAT1; Kuka.VelocityPath=2; Kuka.CurrentCDSetIndex=0; Kuka.MovementParameterFieldEnabled=True; IlfCommand=LIN
;ENDFOLD
$BWDSTART = FALSE
LDAT_ACT = LCPDAT891
FDAT_ACT = FP891
BAS(#CP_PARAMS, 2.0)
SET_CD_PARAMS (0)
LIN XP891
;ENDFOLD

;FOLD LIN P892 Vel=2 m/s CPDAT892 Tool[1]:marker Base[0] ;%{PE}
;FOLD Parameters ;%{h}
;Params IlfProvider=kukaroboter.basistech.inlineforms.movement.old; Kuka.IsGlobalPoint=False; Kuka.PointName=P892; Kuka.BlendingEnabled=False; Kuka.MoveDataName=CPDAT1; Kuka.VelocityPath=2; Kuka.CurrentCDSetIndex=0; Kuka.MovementParameterFieldEnabled=True; IlfCommand=LIN
;ENDFOLD
$BWDSTART = FALSE
LDAT_ACT = LCPDAT892
FDAT_ACT = FP892
BAS(#CP_PARAMS, 2.0)
SET_CD_PARAMS (0)
LIN XP892
;ENDFOLD

;FOLD LIN P893 Vel=2 m/s CPDAT893 Tool[1]:marker Base[0] ;%{PE}
;FOLD Parameters ;%{h}
;Params IlfProvider=kukaroboter.basistech.inlineforms.movement.old; Kuka.IsGlobalPoint=False; Kuka.PointName=P893; Kuka.BlendingEnabled=False; Kuka.MoveDataName=CPDAT1; Kuka.VelocityPath=2; Kuka.CurrentCDSetIndex=0; Kuka.MovementParameterFieldEnabled=True; IlfCommand=LIN
;ENDFOLD
$BWDSTART = FALSE
LDAT_ACT = LCPDAT893
FDAT_ACT = FP893
BAS(#CP_PARAMS, 2.0)
SET_CD_PARAMS (0)
LIN XP893
;ENDFOLD

;FOLD LIN P894 Vel=2 m/s CPDAT894 Tool[1]:marker Base[0] ;%{PE}
;FOLD Parameters ;%{h}
;Params IlfProvider=kukaroboter.basistech.inlineforms.movement.old; Kuka.IsGlobalPoint=False; Kuka.PointName=P894; Kuka.BlendingEnabled=False; Kuka.MoveDataName=CPDAT1; Kuka.VelocityPath=2; Kuka.CurrentCDSetIndex=0; Kuka.MovementParameterFieldEnabled=True; IlfCommand=LIN
;ENDFOLD
$BWDSTART = FALSE
LDAT_ACT = LCPDAT894
FDAT_ACT = FP894
BAS(#CP_PARAMS, 2.0)
SET_CD_PARAMS (0)
LIN XP894
;ENDFOLD

;FOLD LIN P895 Vel=2 m/s CPDAT895 Tool[1]:marker Base[0] ;%{PE}
;FOLD Parameters ;%{h}
;Params IlfProvider=kukaroboter.basistech.inlineforms.movement.old; Kuka.IsGlobalPoint=False; Kuka.PointName=P895; Kuka.BlendingEnabled=False; Kuka.MoveDataName=CPDAT1; Kuka.VelocityPath=2; Kuka.CurrentCDSetIndex=0; Kuka.MovementParameterFieldEnabled=True; IlfCommand=LIN
;ENDFOLD
$BWDSTART = FALSE
LDAT_ACT = LCPDAT895
FDAT_ACT = FP895
BAS(#CP_PARAMS, 2.0)
SET_CD_PARAMS (0)
LIN XP895
;ENDFOLD

;FOLD LIN P896 Vel=2 m/s CPDAT896 Tool[1]:marker Base[0] ;%{PE}
;FOLD Parameters ;%{h}
;Params IlfProvider=kukaroboter.basistech.inlineforms.movement.old; Kuka.IsGlobalPoint=False; Kuka.PointName=P896; Kuka.BlendingEnabled=False; Kuka.MoveDataName=CPDAT1; Kuka.VelocityPath=2; Kuka.CurrentCDSetIndex=0; Kuka.MovementParameterFieldEnabled=True; IlfCommand=LIN
;ENDFOLD
$BWDSTART = FALSE
LDAT_ACT = LCPDAT896
FDAT_ACT = FP896
BAS(#CP_PARAMS, 2.0)
SET_CD_PARAMS (0)
LIN XP896
;ENDFOLD

;FOLD LIN P897 Vel=2 m/s CPDAT897 Tool[1]:marker Base[0] ;%{PE}
;FOLD Parameters ;%{h}
;Params IlfProvider=kukaroboter.basistech.inlineforms.movement.old; Kuka.IsGlobalPoint=False; Kuka.PointName=P897; Kuka.BlendingEnabled=False; Kuka.MoveDataName=CPDAT1; Kuka.VelocityPath=2; Kuka.CurrentCDSetIndex=0; Kuka.MovementParameterFieldEnabled=True; IlfCommand=LIN
;ENDFOLD
$BWDSTART = FALSE
LDAT_ACT = LCPDAT897
FDAT_ACT = FP897
BAS(#CP_PARAMS, 2.0)
SET_CD_PARAMS (0)
LIN XP897
;ENDFOLD

;FOLD LIN P898 Vel=2 m/s CPDAT898 Tool[1]:marker Base[0] ;%{PE}
;FOLD Parameters ;%{h}
;Params IlfProvider=kukaroboter.basistech.inlineforms.movement.old; Kuka.IsGlobalPoint=False; Kuka.PointName=P898; Kuka.BlendingEnabled=False; Kuka.MoveDataName=CPDAT1; Kuka.VelocityPath=2; Kuka.CurrentCDSetIndex=0; Kuka.MovementParameterFieldEnabled=True; IlfCommand=LIN
;ENDFOLD
$BWDSTART = FALSE
LDAT_ACT = LCPDAT898
FDAT_ACT = FP898
BAS(#CP_PARAMS, 2.0)
SET_CD_PARAMS (0)
LIN XP898
;ENDFOLD

;FOLD LIN P899 Vel=2 m/s CPDAT899 Tool[1]:marker Base[0] ;%{PE}
;FOLD Parameters ;%{h}
;Params IlfProvider=kukaroboter.basistech.inlineforms.movement.old; Kuka.IsGlobalPoint=False; Kuka.PointName=P899; Kuka.BlendingEnabled=False; Kuka.MoveDataName=CPDAT1; Kuka.VelocityPath=2; Kuka.CurrentCDSetIndex=0; Kuka.MovementParameterFieldEnabled=True; IlfCommand=LIN
;ENDFOLD
$BWDSTART = FALSE
LDAT_ACT = LCPDAT899
FDAT_ACT = FP899
BAS(#CP_PARAMS, 2.0)
SET_CD_PARAMS (0)
LIN XP899
;ENDFOLD

;FOLD LIN P900 Vel=2 m/s CPDAT900 Tool[1]:marker Base[0] ;%{PE}
;FOLD Parameters ;%{h}
;Params IlfProvider=kukaroboter.basistech.inlineforms.movement.old; Kuka.IsGlobalPoint=False; Kuka.PointName=P900; Kuka.BlendingEnabled=False; Kuka.MoveDataName=CPDAT1; Kuka.VelocityPath=2; Kuka.CurrentCDSetIndex=0; Kuka.MovementParameterFieldEnabled=True; IlfCommand=LIN
;ENDFOLD
$BWDSTART = FALSE
LDAT_ACT = LCPDAT900
FDAT_ACT = FP900
BAS(#CP_PARAMS, 2.0)
SET_CD_PARAMS (0)
LIN XP900
;ENDFOLD

;FOLD LIN P901 Vel=2 m/s CPDAT901 Tool[1]:marker Base[0] ;%{PE}
;FOLD Parameters ;%{h}
;Params IlfProvider=kukaroboter.basistech.inlineforms.movement.old; Kuka.IsGlobalPoint=False; Kuka.PointName=P901; Kuka.BlendingEnabled=False; Kuka.MoveDataName=CPDAT1; Kuka.VelocityPath=2; Kuka.CurrentCDSetIndex=0; Kuka.MovementParameterFieldEnabled=True; IlfCommand=LIN
;ENDFOLD
$BWDSTART = FALSE
LDAT_ACT = LCPDAT901
FDAT_ACT = FP901
BAS(#CP_PARAMS, 2.0)
SET_CD_PARAMS (0)
LIN XP901
;ENDFOLD

;FOLD LIN P902 Vel=2 m/s CPDAT902 Tool[1]:marker Base[0] ;%{PE}
;FOLD Parameters ;%{h}
;Params IlfProvider=kukaroboter.basistech.inlineforms.movement.old; Kuka.IsGlobalPoint=False; Kuka.PointName=P902; Kuka.BlendingEnabled=False; Kuka.MoveDataName=CPDAT1; Kuka.VelocityPath=2; Kuka.CurrentCDSetIndex=0; Kuka.MovementParameterFieldEnabled=True; IlfCommand=LIN
;ENDFOLD
$BWDSTART = FALSE
LDAT_ACT = LCPDAT902
FDAT_ACT = FP902
BAS(#CP_PARAMS, 2.0)
SET_CD_PARAMS (0)
LIN XP902
;ENDFOLD

;FOLD LIN P903 Vel=2 m/s CPDAT903 Tool[1]:marker Base[0] ;%{PE}
;FOLD Parameters ;%{h}
;Params IlfProvider=kukaroboter.basistech.inlineforms.movement.old; Kuka.IsGlobalPoint=False; Kuka.PointName=P903; Kuka.BlendingEnabled=False; Kuka.MoveDataName=CPDAT1; Kuka.VelocityPath=2; Kuka.CurrentCDSetIndex=0; Kuka.MovementParameterFieldEnabled=True; IlfCommand=LIN
;ENDFOLD
$BWDSTART = FALSE
LDAT_ACT = LCPDAT903
FDAT_ACT = FP903
BAS(#CP_PARAMS, 2.0)
SET_CD_PARAMS (0)
LIN XP903
;ENDFOLD

;FOLD LIN P904 Vel=2 m/s CPDAT904 Tool[1]:marker Base[0] ;%{PE}
;FOLD Parameters ;%{h}
;Params IlfProvider=kukaroboter.basistech.inlineforms.movement.old; Kuka.IsGlobalPoint=False; Kuka.PointName=P904; Kuka.BlendingEnabled=False; Kuka.MoveDataName=CPDAT1; Kuka.VelocityPath=2; Kuka.CurrentCDSetIndex=0; Kuka.MovementParameterFieldEnabled=True; IlfCommand=LIN
;ENDFOLD
$BWDSTART = FALSE
LDAT_ACT = LCPDAT904
FDAT_ACT = FP904
BAS(#CP_PARAMS, 2.0)
SET_CD_PARAMS (0)
LIN XP904
;ENDFOLD

;FOLD LIN P905 Vel=2 m/s CPDAT905 Tool[1]:marker Base[0] ;%{PE}
;FOLD Parameters ;%{h}
;Params IlfProvider=kukaroboter.basistech.inlineforms.movement.old; Kuka.IsGlobalPoint=False; Kuka.PointName=P905; Kuka.BlendingEnabled=False; Kuka.MoveDataName=CPDAT1; Kuka.VelocityPath=2; Kuka.CurrentCDSetIndex=0; Kuka.MovementParameterFieldEnabled=True; IlfCommand=LIN
;ENDFOLD
$BWDSTART = FALSE
LDAT_ACT = LCPDAT905
FDAT_ACT = FP905
BAS(#CP_PARAMS, 2.0)
SET_CD_PARAMS (0)
LIN XP905
;ENDFOLD

;FOLD LIN P906 Vel=2 m/s CPDAT906 Tool[1]:marker Base[0] ;%{PE}
;FOLD Parameters ;%{h}
;Params IlfProvider=kukaroboter.basistech.inlineforms.movement.old; Kuka.IsGlobalPoint=False; Kuka.PointName=P906; Kuka.BlendingEnabled=False; Kuka.MoveDataName=CPDAT1; Kuka.VelocityPath=2; Kuka.CurrentCDSetIndex=0; Kuka.MovementParameterFieldEnabled=True; IlfCommand=LIN
;ENDFOLD
$BWDSTART = FALSE
LDAT_ACT = LCPDAT906
FDAT_ACT = FP906
BAS(#CP_PARAMS, 2.0)
SET_CD_PARAMS (0)
LIN XP906
;ENDFOLD

;FOLD LIN P907 Vel=2 m/s CPDAT907 Tool[1]:marker Base[0] ;%{PE}
;FOLD Parameters ;%{h}
;Params IlfProvider=kukaroboter.basistech.inlineforms.movement.old; Kuka.IsGlobalPoint=False; Kuka.PointName=P907; Kuka.BlendingEnabled=False; Kuka.MoveDataName=CPDAT1; Kuka.VelocityPath=2; Kuka.CurrentCDSetIndex=0; Kuka.MovementParameterFieldEnabled=True; IlfCommand=LIN
;ENDFOLD
$BWDSTART = FALSE
LDAT_ACT = LCPDAT907
FDAT_ACT = FP907
BAS(#CP_PARAMS, 2.0)
SET_CD_PARAMS (0)
LIN XP907
;ENDFOLD

;FOLD LIN P908 Vel=2 m/s CPDAT908 Tool[1]:marker Base[0] ;%{PE}
;FOLD Parameters ;%{h}
;Params IlfProvider=kukaroboter.basistech.inlineforms.movement.old; Kuka.IsGlobalPoint=False; Kuka.PointName=P908; Kuka.BlendingEnabled=False; Kuka.MoveDataName=CPDAT1; Kuka.VelocityPath=2; Kuka.CurrentCDSetIndex=0; Kuka.MovementParameterFieldEnabled=True; IlfCommand=LIN
;ENDFOLD
$BWDSTART = FALSE
LDAT_ACT = LCPDAT908
FDAT_ACT = FP908
BAS(#CP_PARAMS, 2.0)
SET_CD_PARAMS (0)
LIN XP908
;ENDFOLD

;FOLD LIN P909 Vel=2 m/s CPDAT909 Tool[1]:marker Base[0] ;%{PE}
;FOLD Parameters ;%{h}
;Params IlfProvider=kukaroboter.basistech.inlineforms.movement.old; Kuka.IsGlobalPoint=False; Kuka.PointName=P909; Kuka.BlendingEnabled=False; Kuka.MoveDataName=CPDAT1; Kuka.VelocityPath=2; Kuka.CurrentCDSetIndex=0; Kuka.MovementParameterFieldEnabled=True; IlfCommand=LIN
;ENDFOLD
$BWDSTART = FALSE
LDAT_ACT = LCPDAT909
FDAT_ACT = FP909
BAS(#CP_PARAMS, 2.0)
SET_CD_PARAMS (0)
LIN XP909
;ENDFOLD

;FOLD LIN P910 Vel=2 m/s CPDAT910 Tool[1]:marker Base[0] ;%{PE}
;FOLD Parameters ;%{h}
;Params IlfProvider=kukaroboter.basistech.inlineforms.movement.old; Kuka.IsGlobalPoint=False; Kuka.PointName=P910; Kuka.BlendingEnabled=False; Kuka.MoveDataName=CPDAT1; Kuka.VelocityPath=2; Kuka.CurrentCDSetIndex=0; Kuka.MovementParameterFieldEnabled=True; IlfCommand=LIN
;ENDFOLD
$BWDSTART = FALSE
LDAT_ACT = LCPDAT910
FDAT_ACT = FP910
BAS(#CP_PARAMS, 2.0)
SET_CD_PARAMS (0)
LIN XP910
;ENDFOLD

;FOLD LIN P911 Vel=2 m/s CPDAT911 Tool[1]:marker Base[0] ;%{PE}
;FOLD Parameters ;%{h}
;Params IlfProvider=kukaroboter.basistech.inlineforms.movement.old; Kuka.IsGlobalPoint=False; Kuka.PointName=P911; Kuka.BlendingEnabled=False; Kuka.MoveDataName=CPDAT1; Kuka.VelocityPath=2; Kuka.CurrentCDSetIndex=0; Kuka.MovementParameterFieldEnabled=True; IlfCommand=LIN
;ENDFOLD
$BWDSTART = FALSE
LDAT_ACT = LCPDAT911
FDAT_ACT = FP911
BAS(#CP_PARAMS, 2.0)
SET_CD_PARAMS (0)
LIN XP911
;ENDFOLD

;FOLD LIN P912 Vel=2 m/s CPDAT912 Tool[1]:marker Base[0] ;%{PE}
;FOLD Parameters ;%{h}
;Params IlfProvider=kukaroboter.basistech.inlineforms.movement.old; Kuka.IsGlobalPoint=False; Kuka.PointName=P912; Kuka.BlendingEnabled=False; Kuka.MoveDataName=CPDAT1; Kuka.VelocityPath=2; Kuka.CurrentCDSetIndex=0; Kuka.MovementParameterFieldEnabled=True; IlfCommand=LIN
;ENDFOLD
$BWDSTART = FALSE
LDAT_ACT = LCPDAT912
FDAT_ACT = FP912
BAS(#CP_PARAMS, 2.0)
SET_CD_PARAMS (0)
LIN XP912
;ENDFOLD

;FOLD LIN P913 Vel=2 m/s CPDAT913 Tool[1]:marker Base[0] ;%{PE}
;FOLD Parameters ;%{h}
;Params IlfProvider=kukaroboter.basistech.inlineforms.movement.old; Kuka.IsGlobalPoint=False; Kuka.PointName=P913; Kuka.BlendingEnabled=False; Kuka.MoveDataName=CPDAT1; Kuka.VelocityPath=2; Kuka.CurrentCDSetIndex=0; Kuka.MovementParameterFieldEnabled=True; IlfCommand=LIN
;ENDFOLD
$BWDSTART = FALSE
LDAT_ACT = LCPDAT913
FDAT_ACT = FP913
BAS(#CP_PARAMS, 2.0)
SET_CD_PARAMS (0)
LIN XP913
;ENDFOLD

;FOLD LIN P914 Vel=2 m/s CPDAT914 Tool[1]:marker Base[0] ;%{PE}
;FOLD Parameters ;%{h}
;Params IlfProvider=kukaroboter.basistech.inlineforms.movement.old; Kuka.IsGlobalPoint=False; Kuka.PointName=P914; Kuka.BlendingEnabled=False; Kuka.MoveDataName=CPDAT1; Kuka.VelocityPath=2; Kuka.CurrentCDSetIndex=0; Kuka.MovementParameterFieldEnabled=True; IlfCommand=LIN
;ENDFOLD
$BWDSTART = FALSE
LDAT_ACT = LCPDAT914
FDAT_ACT = FP914
BAS(#CP_PARAMS, 2.0)
SET_CD_PARAMS (0)
LIN XP914
;ENDFOLD

;FOLD LIN P915 Vel=2 m/s CPDAT915 Tool[1]:marker Base[0] ;%{PE}
;FOLD Parameters ;%{h}
;Params IlfProvider=kukaroboter.basistech.inlineforms.movement.old; Kuka.IsGlobalPoint=False; Kuka.PointName=P915; Kuka.BlendingEnabled=False; Kuka.MoveDataName=CPDAT1; Kuka.VelocityPath=2; Kuka.CurrentCDSetIndex=0; Kuka.MovementParameterFieldEnabled=True; IlfCommand=LIN
;ENDFOLD
$BWDSTART = FALSE
LDAT_ACT = LCPDAT915
FDAT_ACT = FP915
BAS(#CP_PARAMS, 2.0)
SET_CD_PARAMS (0)
LIN XP915
;ENDFOLD

;FOLD LIN P916 Vel=2 m/s CPDAT916 Tool[1]:marker Base[0] ;%{PE}
;FOLD Parameters ;%{h}
;Params IlfProvider=kukaroboter.basistech.inlineforms.movement.old; Kuka.IsGlobalPoint=False; Kuka.PointName=P916; Kuka.BlendingEnabled=False; Kuka.MoveDataName=CPDAT1; Kuka.VelocityPath=2; Kuka.CurrentCDSetIndex=0; Kuka.MovementParameterFieldEnabled=True; IlfCommand=LIN
;ENDFOLD
$BWDSTART = FALSE
LDAT_ACT = LCPDAT916
FDAT_ACT = FP916
BAS(#CP_PARAMS, 2.0)
SET_CD_PARAMS (0)
LIN XP916
;ENDFOLD

;FOLD LIN P917 Vel=2 m/s CPDAT917 Tool[1]:marker Base[0] ;%{PE}
;FOLD Parameters ;%{h}
;Params IlfProvider=kukaroboter.basistech.inlineforms.movement.old; Kuka.IsGlobalPoint=False; Kuka.PointName=P917; Kuka.BlendingEnabled=False; Kuka.MoveDataName=CPDAT1; Kuka.VelocityPath=2; Kuka.CurrentCDSetIndex=0; Kuka.MovementParameterFieldEnabled=True; IlfCommand=LIN
;ENDFOLD
$BWDSTART = FALSE
LDAT_ACT = LCPDAT917
FDAT_ACT = FP917
BAS(#CP_PARAMS, 2.0)
SET_CD_PARAMS (0)
LIN XP917
;ENDFOLD

;FOLD LIN P918 Vel=2 m/s CPDAT918 Tool[1]:marker Base[0] ;%{PE}
;FOLD Parameters ;%{h}
;Params IlfProvider=kukaroboter.basistech.inlineforms.movement.old; Kuka.IsGlobalPoint=False; Kuka.PointName=P918; Kuka.BlendingEnabled=False; Kuka.MoveDataName=CPDAT1; Kuka.VelocityPath=2; Kuka.CurrentCDSetIndex=0; Kuka.MovementParameterFieldEnabled=True; IlfCommand=LIN
;ENDFOLD
$BWDSTART = FALSE
LDAT_ACT = LCPDAT918
FDAT_ACT = FP918
BAS(#CP_PARAMS, 2.0)
SET_CD_PARAMS (0)
LIN XP918
;ENDFOLD

;FOLD LIN P919 Vel=2 m/s CPDAT919 Tool[1]:marker Base[0] ;%{PE}
;FOLD Parameters ;%{h}
;Params IlfProvider=kukaroboter.basistech.inlineforms.movement.old; Kuka.IsGlobalPoint=False; Kuka.PointName=P919; Kuka.BlendingEnabled=False; Kuka.MoveDataName=CPDAT1; Kuka.VelocityPath=2; Kuka.CurrentCDSetIndex=0; Kuka.MovementParameterFieldEnabled=True; IlfCommand=LIN
;ENDFOLD
$BWDSTART = FALSE
LDAT_ACT = LCPDAT919
FDAT_ACT = FP919
BAS(#CP_PARAMS, 2.0)
SET_CD_PARAMS (0)
LIN XP919
;ENDFOLD

;FOLD LIN P920 Vel=2 m/s CPDAT920 Tool[1]:marker Base[0] ;%{PE}
;FOLD Parameters ;%{h}
;Params IlfProvider=kukaroboter.basistech.inlineforms.movement.old; Kuka.IsGlobalPoint=False; Kuka.PointName=P920; Kuka.BlendingEnabled=False; Kuka.MoveDataName=CPDAT1; Kuka.VelocityPath=2; Kuka.CurrentCDSetIndex=0; Kuka.MovementParameterFieldEnabled=True; IlfCommand=LIN
;ENDFOLD
$BWDSTART = FALSE
LDAT_ACT = LCPDAT920
FDAT_ACT = FP920
BAS(#CP_PARAMS, 2.0)
SET_CD_PARAMS (0)
LIN XP920
;ENDFOLD

;FOLD LIN P921 Vel=2 m/s CPDAT921 Tool[1]:marker Base[0] ;%{PE}
;FOLD Parameters ;%{h}
;Params IlfProvider=kukaroboter.basistech.inlineforms.movement.old; Kuka.IsGlobalPoint=False; Kuka.PointName=P921; Kuka.BlendingEnabled=False; Kuka.MoveDataName=CPDAT1; Kuka.VelocityPath=2; Kuka.CurrentCDSetIndex=0; Kuka.MovementParameterFieldEnabled=True; IlfCommand=LIN
;ENDFOLD
$BWDSTART = FALSE
LDAT_ACT = LCPDAT921
FDAT_ACT = FP921
BAS(#CP_PARAMS, 2.0)
SET_CD_PARAMS (0)
LIN XP921
;ENDFOLD

;FOLD LIN P922 Vel=2 m/s CPDAT922 Tool[1]:marker Base[0] ;%{PE}
;FOLD Parameters ;%{h}
;Params IlfProvider=kukaroboter.basistech.inlineforms.movement.old; Kuka.IsGlobalPoint=False; Kuka.PointName=P922; Kuka.BlendingEnabled=False; Kuka.MoveDataName=CPDAT1; Kuka.VelocityPath=2; Kuka.CurrentCDSetIndex=0; Kuka.MovementParameterFieldEnabled=True; IlfCommand=LIN
;ENDFOLD
$BWDSTART = FALSE
LDAT_ACT = LCPDAT922
FDAT_ACT = FP922
BAS(#CP_PARAMS, 2.0)
SET_CD_PARAMS (0)
LIN XP922
;ENDFOLD

;FOLD LIN P923 Vel=2 m/s CPDAT923 Tool[1]:marker Base[0] ;%{PE}
;FOLD Parameters ;%{h}
;Params IlfProvider=kukaroboter.basistech.inlineforms.movement.old; Kuka.IsGlobalPoint=False; Kuka.PointName=P923; Kuka.BlendingEnabled=False; Kuka.MoveDataName=CPDAT1; Kuka.VelocityPath=2; Kuka.CurrentCDSetIndex=0; Kuka.MovementParameterFieldEnabled=True; IlfCommand=LIN
;ENDFOLD
$BWDSTART = FALSE
LDAT_ACT = LCPDAT923
FDAT_ACT = FP923
BAS(#CP_PARAMS, 2.0)
SET_CD_PARAMS (0)
LIN XP923
;ENDFOLD

;FOLD LIN P924 Vel=2 m/s CPDAT924 Tool[1]:marker Base[0] ;%{PE}
;FOLD Parameters ;%{h}
;Params IlfProvider=kukaroboter.basistech.inlineforms.movement.old; Kuka.IsGlobalPoint=False; Kuka.PointName=P924; Kuka.BlendingEnabled=False; Kuka.MoveDataName=CPDAT1; Kuka.VelocityPath=2; Kuka.CurrentCDSetIndex=0; Kuka.MovementParameterFieldEnabled=True; IlfCommand=LIN
;ENDFOLD
$BWDSTART = FALSE
LDAT_ACT = LCPDAT924
FDAT_ACT = FP924
BAS(#CP_PARAMS, 2.0)
SET_CD_PARAMS (0)
LIN XP924
;ENDFOLD

;FOLD LIN P925 Vel=2 m/s CPDAT925 Tool[1]:marker Base[0] ;%{PE}
;FOLD Parameters ;%{h}
;Params IlfProvider=kukaroboter.basistech.inlineforms.movement.old; Kuka.IsGlobalPoint=False; Kuka.PointName=P925; Kuka.BlendingEnabled=False; Kuka.MoveDataName=CPDAT1; Kuka.VelocityPath=2; Kuka.CurrentCDSetIndex=0; Kuka.MovementParameterFieldEnabled=True; IlfCommand=LIN
;ENDFOLD
$BWDSTART = FALSE
LDAT_ACT = LCPDAT925
FDAT_ACT = FP925
BAS(#CP_PARAMS, 2.0)
SET_CD_PARAMS (0)
LIN XP925
;ENDFOLD

;FOLD LIN P926 Vel=2 m/s CPDAT926 Tool[1]:marker Base[0] ;%{PE}
;FOLD Parameters ;%{h}
;Params IlfProvider=kukaroboter.basistech.inlineforms.movement.old; Kuka.IsGlobalPoint=False; Kuka.PointName=P926; Kuka.BlendingEnabled=False; Kuka.MoveDataName=CPDAT1; Kuka.VelocityPath=2; Kuka.CurrentCDSetIndex=0; Kuka.MovementParameterFieldEnabled=True; IlfCommand=LIN
;ENDFOLD
$BWDSTART = FALSE
LDAT_ACT = LCPDAT926
FDAT_ACT = FP926
BAS(#CP_PARAMS, 2.0)
SET_CD_PARAMS (0)
LIN XP926
;ENDFOLD

;FOLD LIN P927 Vel=2 m/s CPDAT927 Tool[1]:marker Base[0] ;%{PE}
;FOLD Parameters ;%{h}
;Params IlfProvider=kukaroboter.basistech.inlineforms.movement.old; Kuka.IsGlobalPoint=False; Kuka.PointName=P927; Kuka.BlendingEnabled=False; Kuka.MoveDataName=CPDAT1; Kuka.VelocityPath=2; Kuka.CurrentCDSetIndex=0; Kuka.MovementParameterFieldEnabled=True; IlfCommand=LIN
;ENDFOLD
$BWDSTART = FALSE
LDAT_ACT = LCPDAT927
FDAT_ACT = FP927
BAS(#CP_PARAMS, 2.0)
SET_CD_PARAMS (0)
LIN XP927
;ENDFOLD

;FOLD LIN P928 Vel=2 m/s CPDAT928 Tool[1]:marker Base[0] ;%{PE}
;FOLD Parameters ;%{h}
;Params IlfProvider=kukaroboter.basistech.inlineforms.movement.old; Kuka.IsGlobalPoint=False; Kuka.PointName=P928; Kuka.BlendingEnabled=False; Kuka.MoveDataName=CPDAT1; Kuka.VelocityPath=2; Kuka.CurrentCDSetIndex=0; Kuka.MovementParameterFieldEnabled=True; IlfCommand=LIN
;ENDFOLD
$BWDSTART = FALSE
LDAT_ACT = LCPDAT928
FDAT_ACT = FP928
BAS(#CP_PARAMS, 2.0)
SET_CD_PARAMS (0)
LIN XP928
;ENDFOLD

;FOLD LIN P929 Vel=2 m/s CPDAT929 Tool[1]:marker Base[0] ;%{PE}
;FOLD Parameters ;%{h}
;Params IlfProvider=kukaroboter.basistech.inlineforms.movement.old; Kuka.IsGlobalPoint=False; Kuka.PointName=P929; Kuka.BlendingEnabled=False; Kuka.MoveDataName=CPDAT1; Kuka.VelocityPath=2; Kuka.CurrentCDSetIndex=0; Kuka.MovementParameterFieldEnabled=True; IlfCommand=LIN
;ENDFOLD
$BWDSTART = FALSE
LDAT_ACT = LCPDAT929
FDAT_ACT = FP929
BAS(#CP_PARAMS, 2.0)
SET_CD_PARAMS (0)
LIN XP929
;ENDFOLD

;FOLD LIN P930 Vel=2 m/s CPDAT930 Tool[1]:marker Base[0] ;%{PE}
;FOLD Parameters ;%{h}
;Params IlfProvider=kukaroboter.basistech.inlineforms.movement.old; Kuka.IsGlobalPoint=False; Kuka.PointName=P930; Kuka.BlendingEnabled=False; Kuka.MoveDataName=CPDAT1; Kuka.VelocityPath=2; Kuka.CurrentCDSetIndex=0; Kuka.MovementParameterFieldEnabled=True; IlfCommand=LIN
;ENDFOLD
$BWDSTART = FALSE
LDAT_ACT = LCPDAT930
FDAT_ACT = FP930
BAS(#CP_PARAMS, 2.0)
SET_CD_PARAMS (0)
LIN XP930
;ENDFOLD

;FOLD LIN P931 Vel=2 m/s CPDAT931 Tool[1]:marker Base[0] ;%{PE}
;FOLD Parameters ;%{h}
;Params IlfProvider=kukaroboter.basistech.inlineforms.movement.old; Kuka.IsGlobalPoint=False; Kuka.PointName=P931; Kuka.BlendingEnabled=False; Kuka.MoveDataName=CPDAT1; Kuka.VelocityPath=2; Kuka.CurrentCDSetIndex=0; Kuka.MovementParameterFieldEnabled=True; IlfCommand=LIN
;ENDFOLD
$BWDSTART = FALSE
LDAT_ACT = LCPDAT931
FDAT_ACT = FP931
BAS(#CP_PARAMS, 2.0)
SET_CD_PARAMS (0)
LIN XP931
;ENDFOLD

;FOLD LIN P932 Vel=2 m/s CPDAT932 Tool[1]:marker Base[0] ;%{PE}
;FOLD Parameters ;%{h}
;Params IlfProvider=kukaroboter.basistech.inlineforms.movement.old; Kuka.IsGlobalPoint=False; Kuka.PointName=P932; Kuka.BlendingEnabled=False; Kuka.MoveDataName=CPDAT1; Kuka.VelocityPath=2; Kuka.CurrentCDSetIndex=0; Kuka.MovementParameterFieldEnabled=True; IlfCommand=LIN
;ENDFOLD
$BWDSTART = FALSE
LDAT_ACT = LCPDAT932
FDAT_ACT = FP932
BAS(#CP_PARAMS, 2.0)
SET_CD_PARAMS (0)
LIN XP932
;ENDFOLD

;FOLD LIN P933 Vel=2 m/s CPDAT933 Tool[1]:marker Base[0] ;%{PE}
;FOLD Parameters ;%{h}
;Params IlfProvider=kukaroboter.basistech.inlineforms.movement.old; Kuka.IsGlobalPoint=False; Kuka.PointName=P933; Kuka.BlendingEnabled=False; Kuka.MoveDataName=CPDAT1; Kuka.VelocityPath=2; Kuka.CurrentCDSetIndex=0; Kuka.MovementParameterFieldEnabled=True; IlfCommand=LIN
;ENDFOLD
$BWDSTART = FALSE
LDAT_ACT = LCPDAT933
FDAT_ACT = FP933
BAS(#CP_PARAMS, 2.0)
SET_CD_PARAMS (0)
LIN XP933
;ENDFOLD

;FOLD LIN P934 Vel=2 m/s CPDAT934 Tool[1]:marker Base[0] ;%{PE}
;FOLD Parameters ;%{h}
;Params IlfProvider=kukaroboter.basistech.inlineforms.movement.old; Kuka.IsGlobalPoint=False; Kuka.PointName=P934; Kuka.BlendingEnabled=False; Kuka.MoveDataName=CPDAT1; Kuka.VelocityPath=2; Kuka.CurrentCDSetIndex=0; Kuka.MovementParameterFieldEnabled=True; IlfCommand=LIN
;ENDFOLD
$BWDSTART = FALSE
LDAT_ACT = LCPDAT934
FDAT_ACT = FP934
BAS(#CP_PARAMS, 2.0)
SET_CD_PARAMS (0)
LIN XP934
;ENDFOLD

;FOLD LIN P935 Vel=2 m/s CPDAT935 Tool[1]:marker Base[0] ;%{PE}
;FOLD Parameters ;%{h}
;Params IlfProvider=kukaroboter.basistech.inlineforms.movement.old; Kuka.IsGlobalPoint=False; Kuka.PointName=P935; Kuka.BlendingEnabled=False; Kuka.MoveDataName=CPDAT1; Kuka.VelocityPath=2; Kuka.CurrentCDSetIndex=0; Kuka.MovementParameterFieldEnabled=True; IlfCommand=LIN
;ENDFOLD
$BWDSTART = FALSE
LDAT_ACT = LCPDAT935
FDAT_ACT = FP935
BAS(#CP_PARAMS, 2.0)
SET_CD_PARAMS (0)
LIN XP935
;ENDFOLD

;FOLD LIN P936 Vel=2 m/s CPDAT936 Tool[1]:marker Base[0] ;%{PE}
;FOLD Parameters ;%{h}
;Params IlfProvider=kukaroboter.basistech.inlineforms.movement.old; Kuka.IsGlobalPoint=False; Kuka.PointName=P936; Kuka.BlendingEnabled=False; Kuka.MoveDataName=CPDAT1; Kuka.VelocityPath=2; Kuka.CurrentCDSetIndex=0; Kuka.MovementParameterFieldEnabled=True; IlfCommand=LIN
;ENDFOLD
$BWDSTART = FALSE
LDAT_ACT = LCPDAT936
FDAT_ACT = FP936
BAS(#CP_PARAMS, 2.0)
SET_CD_PARAMS (0)
LIN XP936
;ENDFOLD

;FOLD LIN P937 Vel=2 m/s CPDAT937 Tool[1]:marker Base[0] ;%{PE}
;FOLD Parameters ;%{h}
;Params IlfProvider=kukaroboter.basistech.inlineforms.movement.old; Kuka.IsGlobalPoint=False; Kuka.PointName=P937; Kuka.BlendingEnabled=False; Kuka.MoveDataName=CPDAT1; Kuka.VelocityPath=2; Kuka.CurrentCDSetIndex=0; Kuka.MovementParameterFieldEnabled=True; IlfCommand=LIN
;ENDFOLD
$BWDSTART = FALSE
LDAT_ACT = LCPDAT937
FDAT_ACT = FP937
BAS(#CP_PARAMS, 2.0)
SET_CD_PARAMS (0)
LIN XP937
;ENDFOLD

;FOLD LIN P938 Vel=2 m/s CPDAT938 Tool[1]:marker Base[0] ;%{PE}
;FOLD Parameters ;%{h}
;Params IlfProvider=kukaroboter.basistech.inlineforms.movement.old; Kuka.IsGlobalPoint=False; Kuka.PointName=P938; Kuka.BlendingEnabled=False; Kuka.MoveDataName=CPDAT1; Kuka.VelocityPath=2; Kuka.CurrentCDSetIndex=0; Kuka.MovementParameterFieldEnabled=True; IlfCommand=LIN
;ENDFOLD
$BWDSTART = FALSE
LDAT_ACT = LCPDAT938
FDAT_ACT = FP938
BAS(#CP_PARAMS, 2.0)
SET_CD_PARAMS (0)
LIN XP938
;ENDFOLD

;FOLD LIN P939 Vel=2 m/s CPDAT939 Tool[1]:marker Base[0] ;%{PE}
;FOLD Parameters ;%{h}
;Params IlfProvider=kukaroboter.basistech.inlineforms.movement.old; Kuka.IsGlobalPoint=False; Kuka.PointName=P939; Kuka.BlendingEnabled=False; Kuka.MoveDataName=CPDAT1; Kuka.VelocityPath=2; Kuka.CurrentCDSetIndex=0; Kuka.MovementParameterFieldEnabled=True; IlfCommand=LIN
;ENDFOLD
$BWDSTART = FALSE
LDAT_ACT = LCPDAT939
FDAT_ACT = FP939
BAS(#CP_PARAMS, 2.0)
SET_CD_PARAMS (0)
LIN XP939
;ENDFOLD

;FOLD LIN P940 Vel=2 m/s CPDAT940 Tool[1]:marker Base[0] ;%{PE}
;FOLD Parameters ;%{h}
;Params IlfProvider=kukaroboter.basistech.inlineforms.movement.old; Kuka.IsGlobalPoint=False; Kuka.PointName=P940; Kuka.BlendingEnabled=False; Kuka.MoveDataName=CPDAT1; Kuka.VelocityPath=2; Kuka.CurrentCDSetIndex=0; Kuka.MovementParameterFieldEnabled=True; IlfCommand=LIN
;ENDFOLD
$BWDSTART = FALSE
LDAT_ACT = LCPDAT940
FDAT_ACT = FP940
BAS(#CP_PARAMS, 2.0)
SET_CD_PARAMS (0)
LIN XP940
;ENDFOLD

;FOLD LIN P941 Vel=2 m/s CPDAT941 Tool[1]:marker Base[0] ;%{PE}
;FOLD Parameters ;%{h}
;Params IlfProvider=kukaroboter.basistech.inlineforms.movement.old; Kuka.IsGlobalPoint=False; Kuka.PointName=P941; Kuka.BlendingEnabled=False; Kuka.MoveDataName=CPDAT1; Kuka.VelocityPath=2; Kuka.CurrentCDSetIndex=0; Kuka.MovementParameterFieldEnabled=True; IlfCommand=LIN
;ENDFOLD
$BWDSTART = FALSE
LDAT_ACT = LCPDAT941
FDAT_ACT = FP941
BAS(#CP_PARAMS, 2.0)
SET_CD_PARAMS (0)
LIN XP941
;ENDFOLD

;FOLD LIN P942 Vel=2 m/s CPDAT942 Tool[1]:marker Base[0] ;%{PE}
;FOLD Parameters ;%{h}
;Params IlfProvider=kukaroboter.basistech.inlineforms.movement.old; Kuka.IsGlobalPoint=False; Kuka.PointName=P942; Kuka.BlendingEnabled=False; Kuka.MoveDataName=CPDAT1; Kuka.VelocityPath=2; Kuka.CurrentCDSetIndex=0; Kuka.MovementParameterFieldEnabled=True; IlfCommand=LIN
;ENDFOLD
$BWDSTART = FALSE
LDAT_ACT = LCPDAT942
FDAT_ACT = FP942
BAS(#CP_PARAMS, 2.0)
SET_CD_PARAMS (0)
LIN XP942
;ENDFOLD

;FOLD LIN P943 Vel=2 m/s CPDAT943 Tool[1]:marker Base[0] ;%{PE}
;FOLD Parameters ;%{h}
;Params IlfProvider=kukaroboter.basistech.inlineforms.movement.old; Kuka.IsGlobalPoint=False; Kuka.PointName=P943; Kuka.BlendingEnabled=False; Kuka.MoveDataName=CPDAT1; Kuka.VelocityPath=2; Kuka.CurrentCDSetIndex=0; Kuka.MovementParameterFieldEnabled=True; IlfCommand=LIN
;ENDFOLD
$BWDSTART = FALSE
LDAT_ACT = LCPDAT943
FDAT_ACT = FP943
BAS(#CP_PARAMS, 2.0)
SET_CD_PARAMS (0)
LIN XP943
;ENDFOLD

;FOLD LIN P944 Vel=2 m/s CPDAT944 Tool[1]:marker Base[0] ;%{PE}
;FOLD Parameters ;%{h}
;Params IlfProvider=kukaroboter.basistech.inlineforms.movement.old; Kuka.IsGlobalPoint=False; Kuka.PointName=P944; Kuka.BlendingEnabled=False; Kuka.MoveDataName=CPDAT1; Kuka.VelocityPath=2; Kuka.CurrentCDSetIndex=0; Kuka.MovementParameterFieldEnabled=True; IlfCommand=LIN
;ENDFOLD
$BWDSTART = FALSE
LDAT_ACT = LCPDAT944
FDAT_ACT = FP944
BAS(#CP_PARAMS, 2.0)
SET_CD_PARAMS (0)
LIN XP944
;ENDFOLD

;FOLD LIN P945 Vel=2 m/s CPDAT945 Tool[1]:marker Base[0] ;%{PE}
;FOLD Parameters ;%{h}
;Params IlfProvider=kukaroboter.basistech.inlineforms.movement.old; Kuka.IsGlobalPoint=False; Kuka.PointName=P945; Kuka.BlendingEnabled=False; Kuka.MoveDataName=CPDAT1; Kuka.VelocityPath=2; Kuka.CurrentCDSetIndex=0; Kuka.MovementParameterFieldEnabled=True; IlfCommand=LIN
;ENDFOLD
$BWDSTART = FALSE
LDAT_ACT = LCPDAT945
FDAT_ACT = FP945
BAS(#CP_PARAMS, 2.0)
SET_CD_PARAMS (0)
LIN XP945
;ENDFOLD

;FOLD LIN P946 Vel=2 m/s CPDAT946 Tool[1]:marker Base[0] ;%{PE}
;FOLD Parameters ;%{h}
;Params IlfProvider=kukaroboter.basistech.inlineforms.movement.old; Kuka.IsGlobalPoint=False; Kuka.PointName=P946; Kuka.BlendingEnabled=False; Kuka.MoveDataName=CPDAT1; Kuka.VelocityPath=2; Kuka.CurrentCDSetIndex=0; Kuka.MovementParameterFieldEnabled=True; IlfCommand=LIN
;ENDFOLD
$BWDSTART = FALSE
LDAT_ACT = LCPDAT946
FDAT_ACT = FP946
BAS(#CP_PARAMS, 2.0)
SET_CD_PARAMS (0)
LIN XP946
;ENDFOLD

;FOLD LIN P947 Vel=2 m/s CPDAT947 Tool[1]:marker Base[0] ;%{PE}
;FOLD Parameters ;%{h}
;Params IlfProvider=kukaroboter.basistech.inlineforms.movement.old; Kuka.IsGlobalPoint=False; Kuka.PointName=P947; Kuka.BlendingEnabled=False; Kuka.MoveDataName=CPDAT1; Kuka.VelocityPath=2; Kuka.CurrentCDSetIndex=0; Kuka.MovementParameterFieldEnabled=True; IlfCommand=LIN
;ENDFOLD
$BWDSTART = FALSE
LDAT_ACT = LCPDAT947
FDAT_ACT = FP947
BAS(#CP_PARAMS, 2.0)
SET_CD_PARAMS (0)
LIN XP947
;ENDFOLD

;FOLD LIN P948 Vel=2 m/s CPDAT948 Tool[1]:marker Base[0] ;%{PE}
;FOLD Parameters ;%{h}
;Params IlfProvider=kukaroboter.basistech.inlineforms.movement.old; Kuka.IsGlobalPoint=False; Kuka.PointName=P948; Kuka.BlendingEnabled=False; Kuka.MoveDataName=CPDAT1; Kuka.VelocityPath=2; Kuka.CurrentCDSetIndex=0; Kuka.MovementParameterFieldEnabled=True; IlfCommand=LIN
;ENDFOLD
$BWDSTART = FALSE
LDAT_ACT = LCPDAT948
FDAT_ACT = FP948
BAS(#CP_PARAMS, 2.0)
SET_CD_PARAMS (0)
LIN XP948
;ENDFOLD

;FOLD LIN P949 Vel=2 m/s CPDAT949 Tool[1]:marker Base[0] ;%{PE}
;FOLD Parameters ;%{h}
;Params IlfProvider=kukaroboter.basistech.inlineforms.movement.old; Kuka.IsGlobalPoint=False; Kuka.PointName=P949; Kuka.BlendingEnabled=False; Kuka.MoveDataName=CPDAT1; Kuka.VelocityPath=2; Kuka.CurrentCDSetIndex=0; Kuka.MovementParameterFieldEnabled=True; IlfCommand=LIN
;ENDFOLD
$BWDSTART = FALSE
LDAT_ACT = LCPDAT949
FDAT_ACT = FP949
BAS(#CP_PARAMS, 2.0)
SET_CD_PARAMS (0)
LIN XP949
;ENDFOLD

;FOLD LIN P950 Vel=2 m/s CPDAT950 Tool[1]:marker Base[0] ;%{PE}
;FOLD Parameters ;%{h}
;Params IlfProvider=kukaroboter.basistech.inlineforms.movement.old; Kuka.IsGlobalPoint=False; Kuka.PointName=P950; Kuka.BlendingEnabled=False; Kuka.MoveDataName=CPDAT1; Kuka.VelocityPath=2; Kuka.CurrentCDSetIndex=0; Kuka.MovementParameterFieldEnabled=True; IlfCommand=LIN
;ENDFOLD
$BWDSTART = FALSE
LDAT_ACT = LCPDAT950
FDAT_ACT = FP950
BAS(#CP_PARAMS, 2.0)
SET_CD_PARAMS (0)
LIN XP950
;ENDFOLD

;FOLD LIN P951 Vel=2 m/s CPDAT951 Tool[1]:marker Base[0] ;%{PE}
;FOLD Parameters ;%{h}
;Params IlfProvider=kukaroboter.basistech.inlineforms.movement.old; Kuka.IsGlobalPoint=False; Kuka.PointName=P951; Kuka.BlendingEnabled=False; Kuka.MoveDataName=CPDAT1; Kuka.VelocityPath=2; Kuka.CurrentCDSetIndex=0; Kuka.MovementParameterFieldEnabled=True; IlfCommand=LIN
;ENDFOLD
$BWDSTART = FALSE
LDAT_ACT = LCPDAT951
FDAT_ACT = FP951
BAS(#CP_PARAMS, 2.0)
SET_CD_PARAMS (0)
LIN XP951
;ENDFOLD

;FOLD LIN P952 Vel=2 m/s CPDAT952 Tool[1]:marker Base[0] ;%{PE}
;FOLD Parameters ;%{h}
;Params IlfProvider=kukaroboter.basistech.inlineforms.movement.old; Kuka.IsGlobalPoint=False; Kuka.PointName=P952; Kuka.BlendingEnabled=False; Kuka.MoveDataName=CPDAT1; Kuka.VelocityPath=2; Kuka.CurrentCDSetIndex=0; Kuka.MovementParameterFieldEnabled=True; IlfCommand=LIN
;ENDFOLD
$BWDSTART = FALSE
LDAT_ACT = LCPDAT952
FDAT_ACT = FP952
BAS(#CP_PARAMS, 2.0)
SET_CD_PARAMS (0)
LIN XP952
;ENDFOLD

;FOLD LIN P953 Vel=2 m/s CPDAT953 Tool[1]:marker Base[0] ;%{PE}
;FOLD Parameters ;%{h}
;Params IlfProvider=kukaroboter.basistech.inlineforms.movement.old; Kuka.IsGlobalPoint=False; Kuka.PointName=P953; Kuka.BlendingEnabled=False; Kuka.MoveDataName=CPDAT1; Kuka.VelocityPath=2; Kuka.CurrentCDSetIndex=0; Kuka.MovementParameterFieldEnabled=True; IlfCommand=LIN
;ENDFOLD
$BWDSTART = FALSE
LDAT_ACT = LCPDAT953
FDAT_ACT = FP953
BAS(#CP_PARAMS, 2.0)
SET_CD_PARAMS (0)
LIN XP953
;ENDFOLD

;FOLD LIN P954 Vel=2 m/s CPDAT954 Tool[1]:marker Base[0] ;%{PE}
;FOLD Parameters ;%{h}
;Params IlfProvider=kukaroboter.basistech.inlineforms.movement.old; Kuka.IsGlobalPoint=False; Kuka.PointName=P954; Kuka.BlendingEnabled=False; Kuka.MoveDataName=CPDAT1; Kuka.VelocityPath=2; Kuka.CurrentCDSetIndex=0; Kuka.MovementParameterFieldEnabled=True; IlfCommand=LIN
;ENDFOLD
$BWDSTART = FALSE
LDAT_ACT = LCPDAT954
FDAT_ACT = FP954
BAS(#CP_PARAMS, 2.0)
SET_CD_PARAMS (0)
LIN XP954
;ENDFOLD

;FOLD LIN P955 Vel=2 m/s CPDAT955 Tool[1]:marker Base[0] ;%{PE}
;FOLD Parameters ;%{h}
;Params IlfProvider=kukaroboter.basistech.inlineforms.movement.old; Kuka.IsGlobalPoint=False; Kuka.PointName=P955; Kuka.BlendingEnabled=False; Kuka.MoveDataName=CPDAT1; Kuka.VelocityPath=2; Kuka.CurrentCDSetIndex=0; Kuka.MovementParameterFieldEnabled=True; IlfCommand=LIN
;ENDFOLD
$BWDSTART = FALSE
LDAT_ACT = LCPDAT955
FDAT_ACT = FP955
BAS(#CP_PARAMS, 2.0)
SET_CD_PARAMS (0)
LIN XP955
;ENDFOLD

;FOLD LIN P956 Vel=2 m/s CPDAT956 Tool[1]:marker Base[0] ;%{PE}
;FOLD Parameters ;%{h}
;Params IlfProvider=kukaroboter.basistech.inlineforms.movement.old; Kuka.IsGlobalPoint=False; Kuka.PointName=P956; Kuka.BlendingEnabled=False; Kuka.MoveDataName=CPDAT1; Kuka.VelocityPath=2; Kuka.CurrentCDSetIndex=0; Kuka.MovementParameterFieldEnabled=True; IlfCommand=LIN
;ENDFOLD
$BWDSTART = FALSE
LDAT_ACT = LCPDAT956
FDAT_ACT = FP956
BAS(#CP_PARAMS, 2.0)
SET_CD_PARAMS (0)
LIN XP956
;ENDFOLD

;FOLD LIN P957 Vel=2 m/s CPDAT957 Tool[1]:marker Base[0] ;%{PE}
;FOLD Parameters ;%{h}
;Params IlfProvider=kukaroboter.basistech.inlineforms.movement.old; Kuka.IsGlobalPoint=False; Kuka.PointName=P957; Kuka.BlendingEnabled=False; Kuka.MoveDataName=CPDAT1; Kuka.VelocityPath=2; Kuka.CurrentCDSetIndex=0; Kuka.MovementParameterFieldEnabled=True; IlfCommand=LIN
;ENDFOLD
$BWDSTART = FALSE
LDAT_ACT = LCPDAT957
FDAT_ACT = FP957
BAS(#CP_PARAMS, 2.0)
SET_CD_PARAMS (0)
LIN XP957
;ENDFOLD

;FOLD LIN P958 Vel=2 m/s CPDAT958 Tool[1]:marker Base[0] ;%{PE}
;FOLD Parameters ;%{h}
;Params IlfProvider=kukaroboter.basistech.inlineforms.movement.old; Kuka.IsGlobalPoint=False; Kuka.PointName=P958; Kuka.BlendingEnabled=False; Kuka.MoveDataName=CPDAT1; Kuka.VelocityPath=2; Kuka.CurrentCDSetIndex=0; Kuka.MovementParameterFieldEnabled=True; IlfCommand=LIN
;ENDFOLD
$BWDSTART = FALSE
LDAT_ACT = LCPDAT958
FDAT_ACT = FP958
BAS(#CP_PARAMS, 2.0)
SET_CD_PARAMS (0)
LIN XP958
;ENDFOLD

;FOLD LIN P959 Vel=2 m/s CPDAT959 Tool[1]:marker Base[0] ;%{PE}
;FOLD Parameters ;%{h}
;Params IlfProvider=kukaroboter.basistech.inlineforms.movement.old; Kuka.IsGlobalPoint=False; Kuka.PointName=P959; Kuka.BlendingEnabled=False; Kuka.MoveDataName=CPDAT1; Kuka.VelocityPath=2; Kuka.CurrentCDSetIndex=0; Kuka.MovementParameterFieldEnabled=True; IlfCommand=LIN
;ENDFOLD
$BWDSTART = FALSE
LDAT_ACT = LCPDAT959
FDAT_ACT = FP959
BAS(#CP_PARAMS, 2.0)
SET_CD_PARAMS (0)
LIN XP959
;ENDFOLD

;FOLD LIN P960 Vel=2 m/s CPDAT960 Tool[1]:marker Base[0] ;%{PE}
;FOLD Parameters ;%{h}
;Params IlfProvider=kukaroboter.basistech.inlineforms.movement.old; Kuka.IsGlobalPoint=False; Kuka.PointName=P960; Kuka.BlendingEnabled=False; Kuka.MoveDataName=CPDAT1; Kuka.VelocityPath=2; Kuka.CurrentCDSetIndex=0; Kuka.MovementParameterFieldEnabled=True; IlfCommand=LIN
;ENDFOLD
$BWDSTART = FALSE
LDAT_ACT = LCPDAT960
FDAT_ACT = FP960
BAS(#CP_PARAMS, 2.0)
SET_CD_PARAMS (0)
LIN XP960
;ENDFOLD

;FOLD LIN P961 Vel=2 m/s CPDAT961 Tool[1]:marker Base[0] ;%{PE}
;FOLD Parameters ;%{h}
;Params IlfProvider=kukaroboter.basistech.inlineforms.movement.old; Kuka.IsGlobalPoint=False; Kuka.PointName=P961; Kuka.BlendingEnabled=False; Kuka.MoveDataName=CPDAT1; Kuka.VelocityPath=2; Kuka.CurrentCDSetIndex=0; Kuka.MovementParameterFieldEnabled=True; IlfCommand=LIN
;ENDFOLD
$BWDSTART = FALSE
LDAT_ACT = LCPDAT961
FDAT_ACT = FP961
BAS(#CP_PARAMS, 2.0)
SET_CD_PARAMS (0)
LIN XP961
;ENDFOLD

;FOLD LIN P962 Vel=2 m/s CPDAT962 Tool[1]:marker Base[0] ;%{PE}
;FOLD Parameters ;%{h}
;Params IlfProvider=kukaroboter.basistech.inlineforms.movement.old; Kuka.IsGlobalPoint=False; Kuka.PointName=P962; Kuka.BlendingEnabled=False; Kuka.MoveDataName=CPDAT1; Kuka.VelocityPath=2; Kuka.CurrentCDSetIndex=0; Kuka.MovementParameterFieldEnabled=True; IlfCommand=LIN
;ENDFOLD
$BWDSTART = FALSE
LDAT_ACT = LCPDAT962
FDAT_ACT = FP962
BAS(#CP_PARAMS, 2.0)
SET_CD_PARAMS (0)
LIN XP962
;ENDFOLD

;FOLD LIN P963 Vel=2 m/s CPDAT963 Tool[1]:marker Base[0] ;%{PE}
;FOLD Parameters ;%{h}
;Params IlfProvider=kukaroboter.basistech.inlineforms.movement.old; Kuka.IsGlobalPoint=False; Kuka.PointName=P963; Kuka.BlendingEnabled=False; Kuka.MoveDataName=CPDAT1; Kuka.VelocityPath=2; Kuka.CurrentCDSetIndex=0; Kuka.MovementParameterFieldEnabled=True; IlfCommand=LIN
;ENDFOLD
$BWDSTART = FALSE
LDAT_ACT = LCPDAT963
FDAT_ACT = FP963
BAS(#CP_PARAMS, 2.0)
SET_CD_PARAMS (0)
LIN XP963
;ENDFOLD

;FOLD LIN P964 Vel=2 m/s CPDAT964 Tool[1]:marker Base[0] ;%{PE}
;FOLD Parameters ;%{h}
;Params IlfProvider=kukaroboter.basistech.inlineforms.movement.old; Kuka.IsGlobalPoint=False; Kuka.PointName=P964; Kuka.BlendingEnabled=False; Kuka.MoveDataName=CPDAT1; Kuka.VelocityPath=2; Kuka.CurrentCDSetIndex=0; Kuka.MovementParameterFieldEnabled=True; IlfCommand=LIN
;ENDFOLD
$BWDSTART = FALSE
LDAT_ACT = LCPDAT964
FDAT_ACT = FP964
BAS(#CP_PARAMS, 2.0)
SET_CD_PARAMS (0)
LIN XP964
;ENDFOLD

;FOLD LIN P965 Vel=2 m/s CPDAT965 Tool[1]:marker Base[0] ;%{PE}
;FOLD Parameters ;%{h}
;Params IlfProvider=kukaroboter.basistech.inlineforms.movement.old; Kuka.IsGlobalPoint=False; Kuka.PointName=P965; Kuka.BlendingEnabled=False; Kuka.MoveDataName=CPDAT1; Kuka.VelocityPath=2; Kuka.CurrentCDSetIndex=0; Kuka.MovementParameterFieldEnabled=True; IlfCommand=LIN
;ENDFOLD
$BWDSTART = FALSE
LDAT_ACT = LCPDAT965
FDAT_ACT = FP965
BAS(#CP_PARAMS, 2.0)
SET_CD_PARAMS (0)
LIN XP965
;ENDFOLD

;FOLD LIN P966 Vel=2 m/s CPDAT966 Tool[1]:marker Base[0] ;%{PE}
;FOLD Parameters ;%{h}
;Params IlfProvider=kukaroboter.basistech.inlineforms.movement.old; Kuka.IsGlobalPoint=False; Kuka.PointName=P966; Kuka.BlendingEnabled=False; Kuka.MoveDataName=CPDAT1; Kuka.VelocityPath=2; Kuka.CurrentCDSetIndex=0; Kuka.MovementParameterFieldEnabled=True; IlfCommand=LIN
;ENDFOLD
$BWDSTART = FALSE
LDAT_ACT = LCPDAT966
FDAT_ACT = FP966
BAS(#CP_PARAMS, 2.0)
SET_CD_PARAMS (0)
LIN XP966
;ENDFOLD

;FOLD LIN P967 Vel=2 m/s CPDAT967 Tool[1]:marker Base[0] ;%{PE}
;FOLD Parameters ;%{h}
;Params IlfProvider=kukaroboter.basistech.inlineforms.movement.old; Kuka.IsGlobalPoint=False; Kuka.PointName=P967; Kuka.BlendingEnabled=False; Kuka.MoveDataName=CPDAT1; Kuka.VelocityPath=2; Kuka.CurrentCDSetIndex=0; Kuka.MovementParameterFieldEnabled=True; IlfCommand=LIN
;ENDFOLD
$BWDSTART = FALSE
LDAT_ACT = LCPDAT967
FDAT_ACT = FP967
BAS(#CP_PARAMS, 2.0)
SET_CD_PARAMS (0)
LIN XP967
;ENDFOLD

;FOLD LIN P968 Vel=2 m/s CPDAT968 Tool[1]:marker Base[0] ;%{PE}
;FOLD Parameters ;%{h}
;Params IlfProvider=kukaroboter.basistech.inlineforms.movement.old; Kuka.IsGlobalPoint=False; Kuka.PointName=P968; Kuka.BlendingEnabled=False; Kuka.MoveDataName=CPDAT1; Kuka.VelocityPath=2; Kuka.CurrentCDSetIndex=0; Kuka.MovementParameterFieldEnabled=True; IlfCommand=LIN
;ENDFOLD
$BWDSTART = FALSE
LDAT_ACT = LCPDAT968
FDAT_ACT = FP968
BAS(#CP_PARAMS, 2.0)
SET_CD_PARAMS (0)
LIN XP968
;ENDFOLD

;FOLD LIN P969 Vel=2 m/s CPDAT969 Tool[1]:marker Base[0] ;%{PE}
;FOLD Parameters ;%{h}
;Params IlfProvider=kukaroboter.basistech.inlineforms.movement.old; Kuka.IsGlobalPoint=False; Kuka.PointName=P969; Kuka.BlendingEnabled=False; Kuka.MoveDataName=CPDAT1; Kuka.VelocityPath=2; Kuka.CurrentCDSetIndex=0; Kuka.MovementParameterFieldEnabled=True; IlfCommand=LIN
;ENDFOLD
$BWDSTART = FALSE
LDAT_ACT = LCPDAT969
FDAT_ACT = FP969
BAS(#CP_PARAMS, 2.0)
SET_CD_PARAMS (0)
LIN XP969
;ENDFOLD

;FOLD LIN P970 Vel=2 m/s CPDAT970 Tool[1]:marker Base[0] ;%{PE}
;FOLD Parameters ;%{h}
;Params IlfProvider=kukaroboter.basistech.inlineforms.movement.old; Kuka.IsGlobalPoint=False; Kuka.PointName=P970; Kuka.BlendingEnabled=False; Kuka.MoveDataName=CPDAT1; Kuka.VelocityPath=2; Kuka.CurrentCDSetIndex=0; Kuka.MovementParameterFieldEnabled=True; IlfCommand=LIN
;ENDFOLD
$BWDSTART = FALSE
LDAT_ACT = LCPDAT970
FDAT_ACT = FP970
BAS(#CP_PARAMS, 2.0)
SET_CD_PARAMS (0)
LIN XP970
;ENDFOLD

;FOLD LIN P971 Vel=2 m/s CPDAT971 Tool[1]:marker Base[0] ;%{PE}
;FOLD Parameters ;%{h}
;Params IlfProvider=kukaroboter.basistech.inlineforms.movement.old; Kuka.IsGlobalPoint=False; Kuka.PointName=P971; Kuka.BlendingEnabled=False; Kuka.MoveDataName=CPDAT1; Kuka.VelocityPath=2; Kuka.CurrentCDSetIndex=0; Kuka.MovementParameterFieldEnabled=True; IlfCommand=LIN
;ENDFOLD
$BWDSTART = FALSE
LDAT_ACT = LCPDAT971
FDAT_ACT = FP971
BAS(#CP_PARAMS, 2.0)
SET_CD_PARAMS (0)
LIN XP971
;ENDFOLD

;FOLD LIN P972 Vel=2 m/s CPDAT972 Tool[1]:marker Base[0] ;%{PE}
;FOLD Parameters ;%{h}
;Params IlfProvider=kukaroboter.basistech.inlineforms.movement.old; Kuka.IsGlobalPoint=False; Kuka.PointName=P972; Kuka.BlendingEnabled=False; Kuka.MoveDataName=CPDAT1; Kuka.VelocityPath=2; Kuka.CurrentCDSetIndex=0; Kuka.MovementParameterFieldEnabled=True; IlfCommand=LIN
;ENDFOLD
$BWDSTART = FALSE
LDAT_ACT = LCPDAT972
FDAT_ACT = FP972
BAS(#CP_PARAMS, 2.0)
SET_CD_PARAMS (0)
LIN XP972
;ENDFOLD

;FOLD LIN P973 Vel=2 m/s CPDAT973 Tool[1]:marker Base[0] ;%{PE}
;FOLD Parameters ;%{h}
;Params IlfProvider=kukaroboter.basistech.inlineforms.movement.old; Kuka.IsGlobalPoint=False; Kuka.PointName=P973; Kuka.BlendingEnabled=False; Kuka.MoveDataName=CPDAT1; Kuka.VelocityPath=2; Kuka.CurrentCDSetIndex=0; Kuka.MovementParameterFieldEnabled=True; IlfCommand=LIN
;ENDFOLD
$BWDSTART = FALSE
LDAT_ACT = LCPDAT973
FDAT_ACT = FP973
BAS(#CP_PARAMS, 2.0)
SET_CD_PARAMS (0)
LIN XP973
;ENDFOLD

;FOLD LIN P974 Vel=2 m/s CPDAT974 Tool[1]:marker Base[0] ;%{PE}
;FOLD Parameters ;%{h}
;Params IlfProvider=kukaroboter.basistech.inlineforms.movement.old; Kuka.IsGlobalPoint=False; Kuka.PointName=P974; Kuka.BlendingEnabled=False; Kuka.MoveDataName=CPDAT1; Kuka.VelocityPath=2; Kuka.CurrentCDSetIndex=0; Kuka.MovementParameterFieldEnabled=True; IlfCommand=LIN
;ENDFOLD
$BWDSTART = FALSE
LDAT_ACT = LCPDAT974
FDAT_ACT = FP974
BAS(#CP_PARAMS, 2.0)
SET_CD_PARAMS (0)
LIN XP974
;ENDFOLD

;FOLD LIN P975 Vel=2 m/s CPDAT975 Tool[1]:marker Base[0] ;%{PE}
;FOLD Parameters ;%{h}
;Params IlfProvider=kukaroboter.basistech.inlineforms.movement.old; Kuka.IsGlobalPoint=False; Kuka.PointName=P975; Kuka.BlendingEnabled=False; Kuka.MoveDataName=CPDAT1; Kuka.VelocityPath=2; Kuka.CurrentCDSetIndex=0; Kuka.MovementParameterFieldEnabled=True; IlfCommand=LIN
;ENDFOLD
$BWDSTART = FALSE
LDAT_ACT = LCPDAT975
FDAT_ACT = FP975
BAS(#CP_PARAMS, 2.0)
SET_CD_PARAMS (0)
LIN XP975
;ENDFOLD

;FOLD LIN P976 Vel=2 m/s CPDAT976 Tool[1]:marker Base[0] ;%{PE}
;FOLD Parameters ;%{h}
;Params IlfProvider=kukaroboter.basistech.inlineforms.movement.old; Kuka.IsGlobalPoint=False; Kuka.PointName=P976; Kuka.BlendingEnabled=False; Kuka.MoveDataName=CPDAT1; Kuka.VelocityPath=2; Kuka.CurrentCDSetIndex=0; Kuka.MovementParameterFieldEnabled=True; IlfCommand=LIN
;ENDFOLD
$BWDSTART = FALSE
LDAT_ACT = LCPDAT976
FDAT_ACT = FP976
BAS(#CP_PARAMS, 2.0)
SET_CD_PARAMS (0)
LIN XP976
;ENDFOLD

;FOLD LIN P977 Vel=2 m/s CPDAT977 Tool[1]:marker Base[0] ;%{PE}
;FOLD Parameters ;%{h}
;Params IlfProvider=kukaroboter.basistech.inlineforms.movement.old; Kuka.IsGlobalPoint=False; Kuka.PointName=P977; Kuka.BlendingEnabled=False; Kuka.MoveDataName=CPDAT1; Kuka.VelocityPath=2; Kuka.CurrentCDSetIndex=0; Kuka.MovementParameterFieldEnabled=True; IlfCommand=LIN
;ENDFOLD
$BWDSTART = FALSE
LDAT_ACT = LCPDAT977
FDAT_ACT = FP977
BAS(#CP_PARAMS, 2.0)
SET_CD_PARAMS (0)
LIN XP977
;ENDFOLD

;FOLD LIN P978 Vel=2 m/s CPDAT978 Tool[1]:marker Base[0] ;%{PE}
;FOLD Parameters ;%{h}
;Params IlfProvider=kukaroboter.basistech.inlineforms.movement.old; Kuka.IsGlobalPoint=False; Kuka.PointName=P978; Kuka.BlendingEnabled=False; Kuka.MoveDataName=CPDAT1; Kuka.VelocityPath=2; Kuka.CurrentCDSetIndex=0; Kuka.MovementParameterFieldEnabled=True; IlfCommand=LIN
;ENDFOLD
$BWDSTART = FALSE
LDAT_ACT = LCPDAT978
FDAT_ACT = FP978
BAS(#CP_PARAMS, 2.0)
SET_CD_PARAMS (0)
LIN XP978
;ENDFOLD

;FOLD LIN P979 Vel=2 m/s CPDAT979 Tool[1]:marker Base[0] ;%{PE}
;FOLD Parameters ;%{h}
;Params IlfProvider=kukaroboter.basistech.inlineforms.movement.old; Kuka.IsGlobalPoint=False; Kuka.PointName=P979; Kuka.BlendingEnabled=False; Kuka.MoveDataName=CPDAT1; Kuka.VelocityPath=2; Kuka.CurrentCDSetIndex=0; Kuka.MovementParameterFieldEnabled=True; IlfCommand=LIN
;ENDFOLD
$BWDSTART = FALSE
LDAT_ACT = LCPDAT979
FDAT_ACT = FP979
BAS(#CP_PARAMS, 2.0)
SET_CD_PARAMS (0)
LIN XP979
;ENDFOLD

;FOLD LIN P980 Vel=2 m/s CPDAT980 Tool[1]:marker Base[0] ;%{PE}
;FOLD Parameters ;%{h}
;Params IlfProvider=kukaroboter.basistech.inlineforms.movement.old; Kuka.IsGlobalPoint=False; Kuka.PointName=P980; Kuka.BlendingEnabled=False; Kuka.MoveDataName=CPDAT1; Kuka.VelocityPath=2; Kuka.CurrentCDSetIndex=0; Kuka.MovementParameterFieldEnabled=True; IlfCommand=LIN
;ENDFOLD
$BWDSTART = FALSE
LDAT_ACT = LCPDAT980
FDAT_ACT = FP980
BAS(#CP_PARAMS, 2.0)
SET_CD_PARAMS (0)
LIN XP980
;ENDFOLD

;FOLD LIN P981 Vel=2 m/s CPDAT981 Tool[1]:marker Base[0] ;%{PE}
;FOLD Parameters ;%{h}
;Params IlfProvider=kukaroboter.basistech.inlineforms.movement.old; Kuka.IsGlobalPoint=False; Kuka.PointName=P981; Kuka.BlendingEnabled=False; Kuka.MoveDataName=CPDAT1; Kuka.VelocityPath=2; Kuka.CurrentCDSetIndex=0; Kuka.MovementParameterFieldEnabled=True; IlfCommand=LIN
;ENDFOLD
$BWDSTART = FALSE
LDAT_ACT = LCPDAT981
FDAT_ACT = FP981
BAS(#CP_PARAMS, 2.0)
SET_CD_PARAMS (0)
LIN XP981
;ENDFOLD

;FOLD LIN P982 Vel=2 m/s CPDAT982 Tool[1]:marker Base[0] ;%{PE}
;FOLD Parameters ;%{h}
;Params IlfProvider=kukaroboter.basistech.inlineforms.movement.old; Kuka.IsGlobalPoint=False; Kuka.PointName=P982; Kuka.BlendingEnabled=False; Kuka.MoveDataName=CPDAT1; Kuka.VelocityPath=2; Kuka.CurrentCDSetIndex=0; Kuka.MovementParameterFieldEnabled=True; IlfCommand=LIN
;ENDFOLD
$BWDSTART = FALSE
LDAT_ACT = LCPDAT982
FDAT_ACT = FP982
BAS(#CP_PARAMS, 2.0)
SET_CD_PARAMS (0)
LIN XP982
;ENDFOLD

;FOLD LIN P983 Vel=2 m/s CPDAT983 Tool[1]:marker Base[0] ;%{PE}
;FOLD Parameters ;%{h}
;Params IlfProvider=kukaroboter.basistech.inlineforms.movement.old; Kuka.IsGlobalPoint=False; Kuka.PointName=P983; Kuka.BlendingEnabled=False; Kuka.MoveDataName=CPDAT1; Kuka.VelocityPath=2; Kuka.CurrentCDSetIndex=0; Kuka.MovementParameterFieldEnabled=True; IlfCommand=LIN
;ENDFOLD
$BWDSTART = FALSE
LDAT_ACT = LCPDAT983
FDAT_ACT = FP983
BAS(#CP_PARAMS, 2.0)
SET_CD_PARAMS (0)
LIN XP983
;ENDFOLD

;FOLD LIN P984 Vel=2 m/s CPDAT984 Tool[1]:marker Base[0] ;%{PE}
;FOLD Parameters ;%{h}
;Params IlfProvider=kukaroboter.basistech.inlineforms.movement.old; Kuka.IsGlobalPoint=False; Kuka.PointName=P984; Kuka.BlendingEnabled=False; Kuka.MoveDataName=CPDAT1; Kuka.VelocityPath=2; Kuka.CurrentCDSetIndex=0; Kuka.MovementParameterFieldEnabled=True; IlfCommand=LIN
;ENDFOLD
$BWDSTART = FALSE
LDAT_ACT = LCPDAT984
FDAT_ACT = FP984
BAS(#CP_PARAMS, 2.0)
SET_CD_PARAMS (0)
LIN XP984
;ENDFOLD

;FOLD LIN P985 Vel=2 m/s CPDAT985 Tool[1]:marker Base[0] ;%{PE}
;FOLD Parameters ;%{h}
;Params IlfProvider=kukaroboter.basistech.inlineforms.movement.old; Kuka.IsGlobalPoint=False; Kuka.PointName=P985; Kuka.BlendingEnabled=False; Kuka.MoveDataName=CPDAT1; Kuka.VelocityPath=2; Kuka.CurrentCDSetIndex=0; Kuka.MovementParameterFieldEnabled=True; IlfCommand=LIN
;ENDFOLD
$BWDSTART = FALSE
LDAT_ACT = LCPDAT985
FDAT_ACT = FP985
BAS(#CP_PARAMS, 2.0)
SET_CD_PARAMS (0)
LIN XP985
;ENDFOLD

;FOLD LIN P986 Vel=2 m/s CPDAT986 Tool[1]:marker Base[0] ;%{PE}
;FOLD Parameters ;%{h}
;Params IlfProvider=kukaroboter.basistech.inlineforms.movement.old; Kuka.IsGlobalPoint=False; Kuka.PointName=P986; Kuka.BlendingEnabled=False; Kuka.MoveDataName=CPDAT1; Kuka.VelocityPath=2; Kuka.CurrentCDSetIndex=0; Kuka.MovementParameterFieldEnabled=True; IlfCommand=LIN
;ENDFOLD
$BWDSTART = FALSE
LDAT_ACT = LCPDAT986
FDAT_ACT = FP986
BAS(#CP_PARAMS, 2.0)
SET_CD_PARAMS (0)
LIN XP986
;ENDFOLD

;FOLD LIN P987 Vel=2 m/s CPDAT987 Tool[1]:marker Base[0] ;%{PE}
;FOLD Parameters ;%{h}
;Params IlfProvider=kukaroboter.basistech.inlineforms.movement.old; Kuka.IsGlobalPoint=False; Kuka.PointName=P987; Kuka.BlendingEnabled=False; Kuka.MoveDataName=CPDAT1; Kuka.VelocityPath=2; Kuka.CurrentCDSetIndex=0; Kuka.MovementParameterFieldEnabled=True; IlfCommand=LIN
;ENDFOLD
$BWDSTART = FALSE
LDAT_ACT = LCPDAT987
FDAT_ACT = FP987
BAS(#CP_PARAMS, 2.0)
SET_CD_PARAMS (0)
LIN XP987
;ENDFOLD

;FOLD LIN P988 Vel=2 m/s CPDAT988 Tool[1]:marker Base[0] ;%{PE}
;FOLD Parameters ;%{h}
;Params IlfProvider=kukaroboter.basistech.inlineforms.movement.old; Kuka.IsGlobalPoint=False; Kuka.PointName=P988; Kuka.BlendingEnabled=False; Kuka.MoveDataName=CPDAT1; Kuka.VelocityPath=2; Kuka.CurrentCDSetIndex=0; Kuka.MovementParameterFieldEnabled=True; IlfCommand=LIN
;ENDFOLD
$BWDSTART = FALSE
LDAT_ACT = LCPDAT988
FDAT_ACT = FP988
BAS(#CP_PARAMS, 2.0)
SET_CD_PARAMS (0)
LIN XP988
;ENDFOLD

;FOLD LIN P989 Vel=2 m/s CPDAT989 Tool[1]:marker Base[0] ;%{PE}
;FOLD Parameters ;%{h}
;Params IlfProvider=kukaroboter.basistech.inlineforms.movement.old; Kuka.IsGlobalPoint=False; Kuka.PointName=P989; Kuka.BlendingEnabled=False; Kuka.MoveDataName=CPDAT1; Kuka.VelocityPath=2; Kuka.CurrentCDSetIndex=0; Kuka.MovementParameterFieldEnabled=True; IlfCommand=LIN
;ENDFOLD
$BWDSTART = FALSE
LDAT_ACT = LCPDAT989
FDAT_ACT = FP989
BAS(#CP_PARAMS, 2.0)
SET_CD_PARAMS (0)
LIN XP989
;ENDFOLD

;FOLD LIN P990 Vel=2 m/s CPDAT990 Tool[1]:marker Base[0] ;%{PE}
;FOLD Parameters ;%{h}
;Params IlfProvider=kukaroboter.basistech.inlineforms.movement.old; Kuka.IsGlobalPoint=False; Kuka.PointName=P990; Kuka.BlendingEnabled=False; Kuka.MoveDataName=CPDAT1; Kuka.VelocityPath=2; Kuka.CurrentCDSetIndex=0; Kuka.MovementParameterFieldEnabled=True; IlfCommand=LIN
;ENDFOLD
$BWDSTART = FALSE
LDAT_ACT = LCPDAT990
FDAT_ACT = FP990
BAS(#CP_PARAMS, 2.0)
SET_CD_PARAMS (0)
LIN XP990
;ENDFOLD

;FOLD LIN P991 Vel=2 m/s CPDAT991 Tool[1]:marker Base[0] ;%{PE}
;FOLD Parameters ;%{h}
;Params IlfProvider=kukaroboter.basistech.inlineforms.movement.old; Kuka.IsGlobalPoint=False; Kuka.PointName=P991; Kuka.BlendingEnabled=False; Kuka.MoveDataName=CPDAT1; Kuka.VelocityPath=2; Kuka.CurrentCDSetIndex=0; Kuka.MovementParameterFieldEnabled=True; IlfCommand=LIN
;ENDFOLD
$BWDSTART = FALSE
LDAT_ACT = LCPDAT991
FDAT_ACT = FP991
BAS(#CP_PARAMS, 2.0)
SET_CD_PARAMS (0)
LIN XP991
;ENDFOLD

;FOLD LIN P992 Vel=2 m/s CPDAT992 Tool[1]:marker Base[0] ;%{PE}
;FOLD Parameters ;%{h}
;Params IlfProvider=kukaroboter.basistech.inlineforms.movement.old; Kuka.IsGlobalPoint=False; Kuka.PointName=P992; Kuka.BlendingEnabled=False; Kuka.MoveDataName=CPDAT1; Kuka.VelocityPath=2; Kuka.CurrentCDSetIndex=0; Kuka.MovementParameterFieldEnabled=True; IlfCommand=LIN
;ENDFOLD
$BWDSTART = FALSE
LDAT_ACT = LCPDAT992
FDAT_ACT = FP992
BAS(#CP_PARAMS, 2.0)
SET_CD_PARAMS (0)
LIN XP992
;ENDFOLD

;FOLD LIN P993 Vel=2 m/s CPDAT993 Tool[1]:marker Base[0] ;%{PE}
;FOLD Parameters ;%{h}
;Params IlfProvider=kukaroboter.basistech.inlineforms.movement.old; Kuka.IsGlobalPoint=False; Kuka.PointName=P993; Kuka.BlendingEnabled=False; Kuka.MoveDataName=CPDAT1; Kuka.VelocityPath=2; Kuka.CurrentCDSetIndex=0; Kuka.MovementParameterFieldEnabled=True; IlfCommand=LIN
;ENDFOLD
$BWDSTART = FALSE
LDAT_ACT = LCPDAT993
FDAT_ACT = FP993
BAS(#CP_PARAMS, 2.0)
SET_CD_PARAMS (0)
LIN XP993
;ENDFOLD

;FOLD LIN P994 Vel=2 m/s CPDAT994 Tool[1]:marker Base[0] ;%{PE}
;FOLD Parameters ;%{h}
;Params IlfProvider=kukaroboter.basistech.inlineforms.movement.old; Kuka.IsGlobalPoint=False; Kuka.PointName=P994; Kuka.BlendingEnabled=False; Kuka.MoveDataName=CPDAT1; Kuka.VelocityPath=2; Kuka.CurrentCDSetIndex=0; Kuka.MovementParameterFieldEnabled=True; IlfCommand=LIN
;ENDFOLD
$BWDSTART = FALSE
LDAT_ACT = LCPDAT994
FDAT_ACT = FP994
BAS(#CP_PARAMS, 2.0)
SET_CD_PARAMS (0)
LIN XP994
;ENDFOLD

;FOLD LIN P995 Vel=2 m/s CPDAT995 Tool[1]:marker Base[0] ;%{PE}
;FOLD Parameters ;%{h}
;Params IlfProvider=kukaroboter.basistech.inlineforms.movement.old; Kuka.IsGlobalPoint=False; Kuka.PointName=P995; Kuka.BlendingEnabled=False; Kuka.MoveDataName=CPDAT1; Kuka.VelocityPath=2; Kuka.CurrentCDSetIndex=0; Kuka.MovementParameterFieldEnabled=True; IlfCommand=LIN
;ENDFOLD
$BWDSTART = FALSE
LDAT_ACT = LCPDAT995
FDAT_ACT = FP995
BAS(#CP_PARAMS, 2.0)
SET_CD_PARAMS (0)
LIN XP995
;ENDFOLD

;FOLD LIN P996 Vel=2 m/s CPDAT996 Tool[1]:marker Base[0] ;%{PE}
;FOLD Parameters ;%{h}
;Params IlfProvider=kukaroboter.basistech.inlineforms.movement.old; Kuka.IsGlobalPoint=False; Kuka.PointName=P996; Kuka.BlendingEnabled=False; Kuka.MoveDataName=CPDAT1; Kuka.VelocityPath=2; Kuka.CurrentCDSetIndex=0; Kuka.MovementParameterFieldEnabled=True; IlfCommand=LIN
;ENDFOLD
$BWDSTART = FALSE
LDAT_ACT = LCPDAT996
FDAT_ACT = FP996
BAS(#CP_PARAMS, 2.0)
SET_CD_PARAMS (0)
LIN XP996
;ENDFOLD

;FOLD LIN P997 Vel=2 m/s CPDAT997 Tool[1]:marker Base[0] ;%{PE}
;FOLD Parameters ;%{h}
;Params IlfProvider=kukaroboter.basistech.inlineforms.movement.old; Kuka.IsGlobalPoint=False; Kuka.PointName=P997; Kuka.BlendingEnabled=False; Kuka.MoveDataName=CPDAT1; Kuka.VelocityPath=2; Kuka.CurrentCDSetIndex=0; Kuka.MovementParameterFieldEnabled=True; IlfCommand=LIN
;ENDFOLD
$BWDSTART = FALSE
LDAT_ACT = LCPDAT997
FDAT_ACT = FP997
BAS(#CP_PARAMS, 2.0)
SET_CD_PARAMS (0)
LIN XP997
;ENDFOLD

;FOLD LIN P998 Vel=2 m/s CPDAT998 Tool[1]:marker Base[0] ;%{PE}
;FOLD Parameters ;%{h}
;Params IlfProvider=kukaroboter.basistech.inlineforms.movement.old; Kuka.IsGlobalPoint=False; Kuka.PointName=P998; Kuka.BlendingEnabled=False; Kuka.MoveDataName=CPDAT1; Kuka.VelocityPath=2; Kuka.CurrentCDSetIndex=0; Kuka.MovementParameterFieldEnabled=True; IlfCommand=LIN
;ENDFOLD
$BWDSTART = FALSE
LDAT_ACT = LCPDAT998
FDAT_ACT = FP998
BAS(#CP_PARAMS, 2.0)
SET_CD_PARAMS (0)
LIN XP998
;ENDFOLD

;FOLD LIN P999 Vel=2 m/s CPDAT999 Tool[1]:marker Base[0] ;%{PE}
;FOLD Parameters ;%{h}
;Params IlfProvider=kukaroboter.basistech.inlineforms.movement.old; Kuka.IsGlobalPoint=False; Kuka.PointName=P999; Kuka.BlendingEnabled=False; Kuka.MoveDataName=CPDAT1; Kuka.VelocityPath=2; Kuka.CurrentCDSetIndex=0; Kuka.MovementParameterFieldEnabled=True; IlfCommand=LIN
;ENDFOLD
$BWDSTART = FALSE
LDAT_ACT = LCPDAT999
FDAT_ACT = FP999
BAS(#CP_PARAMS, 2.0)
SET_CD_PARAMS (0)
LIN XP999
;ENDFOLD

;FOLD LIN P1000 Vel=2 m/s CPDAT1000 Tool[1]:marker Base[0] ;%{PE}
;FOLD Parameters ;%{h}
;Params IlfProvider=kukaroboter.basistech.inlineforms.movement.old; Kuka.IsGlobalPoint=False; Kuka.PointName=P1000; Kuka.BlendingEnabled=False; Kuka.MoveDataName=CPDAT1; Kuka.VelocityPath=2; Kuka.CurrentCDSetIndex=0; Kuka.MovementParameterFieldEnabled=True; IlfCommand=LIN
;ENDFOLD
$BWDSTART = FALSE
LDAT_ACT = LCPDAT1000
FDAT_ACT = FP1000
BAS(#CP_PARAMS, 2.0)
SET_CD_PARAMS (0)
LIN XP1000
;ENDFOLD

;FOLD LIN P1001 Vel=2 m/s CPDAT1001 Tool[1]:marker Base[0] ;%{PE}
;FOLD Parameters ;%{h}
;Params IlfProvider=kukaroboter.basistech.inlineforms.movement.old; Kuka.IsGlobalPoint=False; Kuka.PointName=P1001; Kuka.BlendingEnabled=False; Kuka.MoveDataName=CPDAT1; Kuka.VelocityPath=2; Kuka.CurrentCDSetIndex=0; Kuka.MovementParameterFieldEnabled=True; IlfCommand=LIN
;ENDFOLD
$BWDSTART = FALSE
LDAT_ACT = LCPDAT1001
FDAT_ACT = FP1001
BAS(#CP_PARAMS, 2.0)
SET_CD_PARAMS (0)
LIN XP1001
;ENDFOLD

;FOLD LIN P1002 Vel=2 m/s CPDAT1002 Tool[1]:marker Base[0] ;%{PE}
;FOLD Parameters ;%{h}
;Params IlfProvider=kukaroboter.basistech.inlineforms.movement.old; Kuka.IsGlobalPoint=False; Kuka.PointName=P1002; Kuka.BlendingEnabled=False; Kuka.MoveDataName=CPDAT1; Kuka.VelocityPath=2; Kuka.CurrentCDSetIndex=0; Kuka.MovementParameterFieldEnabled=True; IlfCommand=LIN
;ENDFOLD
$BWDSTART = FALSE
LDAT_ACT = LCPDAT1002
FDAT_ACT = FP1002
BAS(#CP_PARAMS, 2.0)
SET_CD_PARAMS (0)
LIN XP1002
;ENDFOLD

;FOLD LIN P1003 Vel=2 m/s CPDAT1003 Tool[1]:marker Base[0] ;%{PE}
;FOLD Parameters ;%{h}
;Params IlfProvider=kukaroboter.basistech.inlineforms.movement.old; Kuka.IsGlobalPoint=False; Kuka.PointName=P1003; Kuka.BlendingEnabled=False; Kuka.MoveDataName=CPDAT1; Kuka.VelocityPath=2; Kuka.CurrentCDSetIndex=0; Kuka.MovementParameterFieldEnabled=True; IlfCommand=LIN
;ENDFOLD
$BWDSTART = FALSE
LDAT_ACT = LCPDAT1003
FDAT_ACT = FP1003
BAS(#CP_PARAMS, 2.0)
SET_CD_PARAMS (0)
LIN XP1003
;ENDFOLD

;FOLD LIN P1004 Vel=2 m/s CPDAT1004 Tool[1]:marker Base[0] ;%{PE}
;FOLD Parameters ;%{h}
;Params IlfProvider=kukaroboter.basistech.inlineforms.movement.old; Kuka.IsGlobalPoint=False; Kuka.PointName=P1004; Kuka.BlendingEnabled=False; Kuka.MoveDataName=CPDAT1; Kuka.VelocityPath=2; Kuka.CurrentCDSetIndex=0; Kuka.MovementParameterFieldEnabled=True; IlfCommand=LIN
;ENDFOLD
$BWDSTART = FALSE
LDAT_ACT = LCPDAT1004
FDAT_ACT = FP1004
BAS(#CP_PARAMS, 2.0)
SET_CD_PARAMS (0)
LIN XP1004
;ENDFOLD

;FOLD LIN P1005 Vel=2 m/s CPDAT1005 Tool[1]:marker Base[0] ;%{PE}
;FOLD Parameters ;%{h}
;Params IlfProvider=kukaroboter.basistech.inlineforms.movement.old; Kuka.IsGlobalPoint=False; Kuka.PointName=P1005; Kuka.BlendingEnabled=False; Kuka.MoveDataName=CPDAT1; Kuka.VelocityPath=2; Kuka.CurrentCDSetIndex=0; Kuka.MovementParameterFieldEnabled=True; IlfCommand=LIN
;ENDFOLD
$BWDSTART = FALSE
LDAT_ACT = LCPDAT1005
FDAT_ACT = FP1005
BAS(#CP_PARAMS, 2.0)
SET_CD_PARAMS (0)
LIN XP1005
;ENDFOLD

;FOLD LIN P1006 Vel=2 m/s CPDAT1006 Tool[1]:marker Base[0] ;%{PE}
;FOLD Parameters ;%{h}
;Params IlfProvider=kukaroboter.basistech.inlineforms.movement.old; Kuka.IsGlobalPoint=False; Kuka.PointName=P1006; Kuka.BlendingEnabled=False; Kuka.MoveDataName=CPDAT1; Kuka.VelocityPath=2; Kuka.CurrentCDSetIndex=0; Kuka.MovementParameterFieldEnabled=True; IlfCommand=LIN
;ENDFOLD
$BWDSTART = FALSE
LDAT_ACT = LCPDAT1006
FDAT_ACT = FP1006
BAS(#CP_PARAMS, 2.0)
SET_CD_PARAMS (0)
LIN XP1006
;ENDFOLD

;FOLD LIN P1007 Vel=2 m/s CPDAT1007 Tool[1]:marker Base[0] ;%{PE}
;FOLD Parameters ;%{h}
;Params IlfProvider=kukaroboter.basistech.inlineforms.movement.old; Kuka.IsGlobalPoint=False; Kuka.PointName=P1007; Kuka.BlendingEnabled=False; Kuka.MoveDataName=CPDAT1; Kuka.VelocityPath=2; Kuka.CurrentCDSetIndex=0; Kuka.MovementParameterFieldEnabled=True; IlfCommand=LIN
;ENDFOLD
$BWDSTART = FALSE
LDAT_ACT = LCPDAT1007
FDAT_ACT = FP1007
BAS(#CP_PARAMS, 2.0)
SET_CD_PARAMS (0)
LIN XP1007
;ENDFOLD

;FOLD LIN P1008 Vel=2 m/s CPDAT1008 Tool[1]:marker Base[0] ;%{PE}
;FOLD Parameters ;%{h}
;Params IlfProvider=kukaroboter.basistech.inlineforms.movement.old; Kuka.IsGlobalPoint=False; Kuka.PointName=P1008; Kuka.BlendingEnabled=False; Kuka.MoveDataName=CPDAT1; Kuka.VelocityPath=2; Kuka.CurrentCDSetIndex=0; Kuka.MovementParameterFieldEnabled=True; IlfCommand=LIN
;ENDFOLD
$BWDSTART = FALSE
LDAT_ACT = LCPDAT1008
FDAT_ACT = FP1008
BAS(#CP_PARAMS, 2.0)
SET_CD_PARAMS (0)
LIN XP1008
;ENDFOLD

;FOLD LIN P1009 Vel=2 m/s CPDAT1009 Tool[1]:marker Base[0] ;%{PE}
;FOLD Parameters ;%{h}
;Params IlfProvider=kukaroboter.basistech.inlineforms.movement.old; Kuka.IsGlobalPoint=False; Kuka.PointName=P1009; Kuka.BlendingEnabled=False; Kuka.MoveDataName=CPDAT1; Kuka.VelocityPath=2; Kuka.CurrentCDSetIndex=0; Kuka.MovementParameterFieldEnabled=True; IlfCommand=LIN
;ENDFOLD
$BWDSTART = FALSE
LDAT_ACT = LCPDAT1009
FDAT_ACT = FP1009
BAS(#CP_PARAMS, 2.0)
SET_CD_PARAMS (0)
LIN XP1009
;ENDFOLD

;FOLD LIN P1010 Vel=2 m/s CPDAT1010 Tool[1]:marker Base[0] ;%{PE}
;FOLD Parameters ;%{h}
;Params IlfProvider=kukaroboter.basistech.inlineforms.movement.old; Kuka.IsGlobalPoint=False; Kuka.PointName=P1010; Kuka.BlendingEnabled=False; Kuka.MoveDataName=CPDAT1; Kuka.VelocityPath=2; Kuka.CurrentCDSetIndex=0; Kuka.MovementParameterFieldEnabled=True; IlfCommand=LIN
;ENDFOLD
$BWDSTART = FALSE
LDAT_ACT = LCPDAT1010
FDAT_ACT = FP1010
BAS(#CP_PARAMS, 2.0)
SET_CD_PARAMS (0)
LIN XP1010
;ENDFOLD

;FOLD LIN P1011 Vel=2 m/s CPDAT1011 Tool[1]:marker Base[0] ;%{PE}
;FOLD Parameters ;%{h}
;Params IlfProvider=kukaroboter.basistech.inlineforms.movement.old; Kuka.IsGlobalPoint=False; Kuka.PointName=P1011; Kuka.BlendingEnabled=False; Kuka.MoveDataName=CPDAT1; Kuka.VelocityPath=2; Kuka.CurrentCDSetIndex=0; Kuka.MovementParameterFieldEnabled=True; IlfCommand=LIN
;ENDFOLD
$BWDSTART = FALSE
LDAT_ACT = LCPDAT1011
FDAT_ACT = FP1011
BAS(#CP_PARAMS, 2.0)
SET_CD_PARAMS (0)
LIN XP1011
;ENDFOLD

;FOLD LIN P1012 Vel=2 m/s CPDAT1012 Tool[1]:marker Base[0] ;%{PE}
;FOLD Parameters ;%{h}
;Params IlfProvider=kukaroboter.basistech.inlineforms.movement.old; Kuka.IsGlobalPoint=False; Kuka.PointName=P1012; Kuka.BlendingEnabled=False; Kuka.MoveDataName=CPDAT1; Kuka.VelocityPath=2; Kuka.CurrentCDSetIndex=0; Kuka.MovementParameterFieldEnabled=True; IlfCommand=LIN
;ENDFOLD
$BWDSTART = FALSE
LDAT_ACT = LCPDAT1012
FDAT_ACT = FP1012
BAS(#CP_PARAMS, 2.0)
SET_CD_PARAMS (0)
LIN XP1012
;ENDFOLD

;FOLD LIN P1013 Vel=2 m/s CPDAT1013 Tool[1]:marker Base[0] ;%{PE}
;FOLD Parameters ;%{h}
;Params IlfProvider=kukaroboter.basistech.inlineforms.movement.old; Kuka.IsGlobalPoint=False; Kuka.PointName=P1013; Kuka.BlendingEnabled=False; Kuka.MoveDataName=CPDAT1; Kuka.VelocityPath=2; Kuka.CurrentCDSetIndex=0; Kuka.MovementParameterFieldEnabled=True; IlfCommand=LIN
;ENDFOLD
$BWDSTART = FALSE
LDAT_ACT = LCPDAT1013
FDAT_ACT = FP1013
BAS(#CP_PARAMS, 2.0)
SET_CD_PARAMS (0)
LIN XP1013
;ENDFOLD

;FOLD LIN P1014 Vel=2 m/s CPDAT1014 Tool[1]:marker Base[0] ;%{PE}
;FOLD Parameters ;%{h}
;Params IlfProvider=kukaroboter.basistech.inlineforms.movement.old; Kuka.IsGlobalPoint=False; Kuka.PointName=P1014; Kuka.BlendingEnabled=False; Kuka.MoveDataName=CPDAT1; Kuka.VelocityPath=2; Kuka.CurrentCDSetIndex=0; Kuka.MovementParameterFieldEnabled=True; IlfCommand=LIN
;ENDFOLD
$BWDSTART = FALSE
LDAT_ACT = LCPDAT1014
FDAT_ACT = FP1014
BAS(#CP_PARAMS, 2.0)
SET_CD_PARAMS (0)
LIN XP1014
;ENDFOLD

;FOLD LIN P1015 Vel=2 m/s CPDAT1015 Tool[1]:marker Base[0] ;%{PE}
;FOLD Parameters ;%{h}
;Params IlfProvider=kukaroboter.basistech.inlineforms.movement.old; Kuka.IsGlobalPoint=False; Kuka.PointName=P1015; Kuka.BlendingEnabled=False; Kuka.MoveDataName=CPDAT1; Kuka.VelocityPath=2; Kuka.CurrentCDSetIndex=0; Kuka.MovementParameterFieldEnabled=True; IlfCommand=LIN
;ENDFOLD
$BWDSTART = FALSE
LDAT_ACT = LCPDAT1015
FDAT_ACT = FP1015
BAS(#CP_PARAMS, 2.0)
SET_CD_PARAMS (0)
LIN XP1015
;ENDFOLD

;FOLD LIN P1016 Vel=2 m/s CPDAT1016 Tool[1]:marker Base[0] ;%{PE}
;FOLD Parameters ;%{h}
;Params IlfProvider=kukaroboter.basistech.inlineforms.movement.old; Kuka.IsGlobalPoint=False; Kuka.PointName=P1016; Kuka.BlendingEnabled=False; Kuka.MoveDataName=CPDAT1; Kuka.VelocityPath=2; Kuka.CurrentCDSetIndex=0; Kuka.MovementParameterFieldEnabled=True; IlfCommand=LIN
;ENDFOLD
$BWDSTART = FALSE
LDAT_ACT = LCPDAT1016
FDAT_ACT = FP1016
BAS(#CP_PARAMS, 2.0)
SET_CD_PARAMS (0)
LIN XP1016
;ENDFOLD

;FOLD LIN P1017 Vel=2 m/s CPDAT1017 Tool[1]:marker Base[0] ;%{PE}
;FOLD Parameters ;%{h}
;Params IlfProvider=kukaroboter.basistech.inlineforms.movement.old; Kuka.IsGlobalPoint=False; Kuka.PointName=P1017; Kuka.BlendingEnabled=False; Kuka.MoveDataName=CPDAT1; Kuka.VelocityPath=2; Kuka.CurrentCDSetIndex=0; Kuka.MovementParameterFieldEnabled=True; IlfCommand=LIN
;ENDFOLD
$BWDSTART = FALSE
LDAT_ACT = LCPDAT1017
FDAT_ACT = FP1017
BAS(#CP_PARAMS, 2.0)
SET_CD_PARAMS (0)
LIN XP1017
;ENDFOLD

;FOLD LIN P1018 Vel=2 m/s CPDAT1018 Tool[1]:marker Base[0] ;%{PE}
;FOLD Parameters ;%{h}
;Params IlfProvider=kukaroboter.basistech.inlineforms.movement.old; Kuka.IsGlobalPoint=False; Kuka.PointName=P1018; Kuka.BlendingEnabled=False; Kuka.MoveDataName=CPDAT1; Kuka.VelocityPath=2; Kuka.CurrentCDSetIndex=0; Kuka.MovementParameterFieldEnabled=True; IlfCommand=LIN
;ENDFOLD
$BWDSTART = FALSE
LDAT_ACT = LCPDAT1018
FDAT_ACT = FP1018
BAS(#CP_PARAMS, 2.0)
SET_CD_PARAMS (0)
LIN XP1018
;ENDFOLD

;FOLD LIN P1019 Vel=2 m/s CPDAT1019 Tool[1]:marker Base[0] ;%{PE}
;FOLD Parameters ;%{h}
;Params IlfProvider=kukaroboter.basistech.inlineforms.movement.old; Kuka.IsGlobalPoint=False; Kuka.PointName=P1019; Kuka.BlendingEnabled=False; Kuka.MoveDataName=CPDAT1; Kuka.VelocityPath=2; Kuka.CurrentCDSetIndex=0; Kuka.MovementParameterFieldEnabled=True; IlfCommand=LIN
;ENDFOLD
$BWDSTART = FALSE
LDAT_ACT = LCPDAT1019
FDAT_ACT = FP1019
BAS(#CP_PARAMS, 2.0)
SET_CD_PARAMS (0)
LIN XP1019
;ENDFOLD

;FOLD LIN P1020 Vel=2 m/s CPDAT1020 Tool[1]:marker Base[0] ;%{PE}
;FOLD Parameters ;%{h}
;Params IlfProvider=kukaroboter.basistech.inlineforms.movement.old; Kuka.IsGlobalPoint=False; Kuka.PointName=P1020; Kuka.BlendingEnabled=False; Kuka.MoveDataName=CPDAT1; Kuka.VelocityPath=2; Kuka.CurrentCDSetIndex=0; Kuka.MovementParameterFieldEnabled=True; IlfCommand=LIN
;ENDFOLD
$BWDSTART = FALSE
LDAT_ACT = LCPDAT1020
FDAT_ACT = FP1020
BAS(#CP_PARAMS, 2.0)
SET_CD_PARAMS (0)
LIN XP1020
;ENDFOLD

;FOLD LIN P1021 Vel=2 m/s CPDAT1021 Tool[1]:marker Base[0] ;%{PE}
;FOLD Parameters ;%{h}
;Params IlfProvider=kukaroboter.basistech.inlineforms.movement.old; Kuka.IsGlobalPoint=False; Kuka.PointName=P1021; Kuka.BlendingEnabled=False; Kuka.MoveDataName=CPDAT1; Kuka.VelocityPath=2; Kuka.CurrentCDSetIndex=0; Kuka.MovementParameterFieldEnabled=True; IlfCommand=LIN
;ENDFOLD
$BWDSTART = FALSE
LDAT_ACT = LCPDAT1021
FDAT_ACT = FP1021
BAS(#CP_PARAMS, 2.0)
SET_CD_PARAMS (0)
LIN XP1021
;ENDFOLD

;FOLD LIN P1022 Vel=2 m/s CPDAT1022 Tool[1]:marker Base[0] ;%{PE}
;FOLD Parameters ;%{h}
;Params IlfProvider=kukaroboter.basistech.inlineforms.movement.old; Kuka.IsGlobalPoint=False; Kuka.PointName=P1022; Kuka.BlendingEnabled=False; Kuka.MoveDataName=CPDAT1; Kuka.VelocityPath=2; Kuka.CurrentCDSetIndex=0; Kuka.MovementParameterFieldEnabled=True; IlfCommand=LIN
;ENDFOLD
$BWDSTART = FALSE
LDAT_ACT = LCPDAT1022
FDAT_ACT = FP1022
BAS(#CP_PARAMS, 2.0)
SET_CD_PARAMS (0)
LIN XP1022
;ENDFOLD

;FOLD LIN P1023 Vel=2 m/s CPDAT1023 Tool[1]:marker Base[0] ;%{PE}
;FOLD Parameters ;%{h}
;Params IlfProvider=kukaroboter.basistech.inlineforms.movement.old; Kuka.IsGlobalPoint=False; Kuka.PointName=P1023; Kuka.BlendingEnabled=False; Kuka.MoveDataName=CPDAT1; Kuka.VelocityPath=2; Kuka.CurrentCDSetIndex=0; Kuka.MovementParameterFieldEnabled=True; IlfCommand=LIN
;ENDFOLD
$BWDSTART = FALSE
LDAT_ACT = LCPDAT1023
FDAT_ACT = FP1023
BAS(#CP_PARAMS, 2.0)
SET_CD_PARAMS (0)
LIN XP1023
;ENDFOLD

;FOLD LIN P1024 Vel=2 m/s CPDAT1024 Tool[1]:marker Base[0] ;%{PE}
;FOLD Parameters ;%{h}
;Params IlfProvider=kukaroboter.basistech.inlineforms.movement.old; Kuka.IsGlobalPoint=False; Kuka.PointName=P1024; Kuka.BlendingEnabled=False; Kuka.MoveDataName=CPDAT1; Kuka.VelocityPath=2; Kuka.CurrentCDSetIndex=0; Kuka.MovementParameterFieldEnabled=True; IlfCommand=LIN
;ENDFOLD
$BWDSTART = FALSE
LDAT_ACT = LCPDAT1024
FDAT_ACT = FP1024
BAS(#CP_PARAMS, 2.0)
SET_CD_PARAMS (0)
LIN XP1024
;ENDFOLD

;FOLD LIN P1025 Vel=2 m/s CPDAT1025 Tool[1]:marker Base[0] ;%{PE}
;FOLD Parameters ;%{h}
;Params IlfProvider=kukaroboter.basistech.inlineforms.movement.old; Kuka.IsGlobalPoint=False; Kuka.PointName=P1025; Kuka.BlendingEnabled=False; Kuka.MoveDataName=CPDAT1; Kuka.VelocityPath=2; Kuka.CurrentCDSetIndex=0; Kuka.MovementParameterFieldEnabled=True; IlfCommand=LIN
;ENDFOLD
$BWDSTART = FALSE
LDAT_ACT = LCPDAT1025
FDAT_ACT = FP1025
BAS(#CP_PARAMS, 2.0)
SET_CD_PARAMS (0)
LIN XP1025
;ENDFOLD

;FOLD LIN P1026 Vel=2 m/s CPDAT1026 Tool[1]:marker Base[0] ;%{PE}
;FOLD Parameters ;%{h}
;Params IlfProvider=kukaroboter.basistech.inlineforms.movement.old; Kuka.IsGlobalPoint=False; Kuka.PointName=P1026; Kuka.BlendingEnabled=False; Kuka.MoveDataName=CPDAT1; Kuka.VelocityPath=2; Kuka.CurrentCDSetIndex=0; Kuka.MovementParameterFieldEnabled=True; IlfCommand=LIN
;ENDFOLD
$BWDSTART = FALSE
LDAT_ACT = LCPDAT1026
FDAT_ACT = FP1026
BAS(#CP_PARAMS, 2.0)
SET_CD_PARAMS (0)
LIN XP1026
;ENDFOLD

;FOLD LIN P1027 Vel=2 m/s CPDAT1027 Tool[1]:marker Base[0] ;%{PE}
;FOLD Parameters ;%{h}
;Params IlfProvider=kukaroboter.basistech.inlineforms.movement.old; Kuka.IsGlobalPoint=False; Kuka.PointName=P1027; Kuka.BlendingEnabled=False; Kuka.MoveDataName=CPDAT1; Kuka.VelocityPath=2; Kuka.CurrentCDSetIndex=0; Kuka.MovementParameterFieldEnabled=True; IlfCommand=LIN
;ENDFOLD
$BWDSTART = FALSE
LDAT_ACT = LCPDAT1027
FDAT_ACT = FP1027
BAS(#CP_PARAMS, 2.0)
SET_CD_PARAMS (0)
LIN XP1027
;ENDFOLD

;FOLD LIN P1028 Vel=2 m/s CPDAT1028 Tool[1]:marker Base[0] ;%{PE}
;FOLD Parameters ;%{h}
;Params IlfProvider=kukaroboter.basistech.inlineforms.movement.old; Kuka.IsGlobalPoint=False; Kuka.PointName=P1028; Kuka.BlendingEnabled=False; Kuka.MoveDataName=CPDAT1; Kuka.VelocityPath=2; Kuka.CurrentCDSetIndex=0; Kuka.MovementParameterFieldEnabled=True; IlfCommand=LIN
;ENDFOLD
$BWDSTART = FALSE
LDAT_ACT = LCPDAT1028
FDAT_ACT = FP1028
BAS(#CP_PARAMS, 2.0)
SET_CD_PARAMS (0)
LIN XP1028
;ENDFOLD

;FOLD LIN P1029 Vel=2 m/s CPDAT1029 Tool[1]:marker Base[0] ;%{PE}
;FOLD Parameters ;%{h}
;Params IlfProvider=kukaroboter.basistech.inlineforms.movement.old; Kuka.IsGlobalPoint=False; Kuka.PointName=P1029; Kuka.BlendingEnabled=False; Kuka.MoveDataName=CPDAT1; Kuka.VelocityPath=2; Kuka.CurrentCDSetIndex=0; Kuka.MovementParameterFieldEnabled=True; IlfCommand=LIN
;ENDFOLD
$BWDSTART = FALSE
LDAT_ACT = LCPDAT1029
FDAT_ACT = FP1029
BAS(#CP_PARAMS, 2.0)
SET_CD_PARAMS (0)
LIN XP1029
;ENDFOLD

;FOLD LIN P1030 Vel=2 m/s CPDAT1030 Tool[1]:marker Base[0] ;%{PE}
;FOLD Parameters ;%{h}
;Params IlfProvider=kukaroboter.basistech.inlineforms.movement.old; Kuka.IsGlobalPoint=False; Kuka.PointName=P1030; Kuka.BlendingEnabled=False; Kuka.MoveDataName=CPDAT1; Kuka.VelocityPath=2; Kuka.CurrentCDSetIndex=0; Kuka.MovementParameterFieldEnabled=True; IlfCommand=LIN
;ENDFOLD
$BWDSTART = FALSE
LDAT_ACT = LCPDAT1030
FDAT_ACT = FP1030
BAS(#CP_PARAMS, 2.0)
SET_CD_PARAMS (0)
LIN XP1030
;ENDFOLD

;FOLD LIN P1031 Vel=2 m/s CPDAT1031 Tool[1]:marker Base[0] ;%{PE}
;FOLD Parameters ;%{h}
;Params IlfProvider=kukaroboter.basistech.inlineforms.movement.old; Kuka.IsGlobalPoint=False; Kuka.PointName=P1031; Kuka.BlendingEnabled=False; Kuka.MoveDataName=CPDAT1; Kuka.VelocityPath=2; Kuka.CurrentCDSetIndex=0; Kuka.MovementParameterFieldEnabled=True; IlfCommand=LIN
;ENDFOLD
$BWDSTART = FALSE
LDAT_ACT = LCPDAT1031
FDAT_ACT = FP1031
BAS(#CP_PARAMS, 2.0)
SET_CD_PARAMS (0)
LIN XP1031
;ENDFOLD

;FOLD LIN P1032 Vel=2 m/s CPDAT1032 Tool[1]:marker Base[0] ;%{PE}
;FOLD Parameters ;%{h}
;Params IlfProvider=kukaroboter.basistech.inlineforms.movement.old; Kuka.IsGlobalPoint=False; Kuka.PointName=P1032; Kuka.BlendingEnabled=False; Kuka.MoveDataName=CPDAT1; Kuka.VelocityPath=2; Kuka.CurrentCDSetIndex=0; Kuka.MovementParameterFieldEnabled=True; IlfCommand=LIN
;ENDFOLD
$BWDSTART = FALSE
LDAT_ACT = LCPDAT1032
FDAT_ACT = FP1032
BAS(#CP_PARAMS, 2.0)
SET_CD_PARAMS (0)
LIN XP1032
;ENDFOLD

